// TIA Portal project "R1A-Cabi" (V15)

(* hardware
DEVICE "LINHA-DENIN"  ET 200S station
   slot 0: "Rack 0"  Rail
   slot 2: "IM151-8 PN/DP CPU"  IM151-8 CPU  6ES7 151-8AB00-0AB0  V2.7
      slot 1: "PROFINET-SLAVE"  PN-IO
         slot 1: "Port_1"  Port
         slot 2: "Port_2"  Port
         slot 3: "Port_3"  Port
   slot 4: "PM-E 24VDC_1"  PM-E 24VDC  6ES7 138-4CA01-0AA0
   slot 5: "DP interface_1"  DP  6ES7 138-4HA00-0AB0  V1.0
   slot 5: "8DI x 24VDC_1"  8DI x 24VDC  6ES7 131-4BF00-0AA0
   slot 6: "8DI x 24VDC_2"  8DI x 24VDC  6ES7 131-4BF00-0AA0
   slot 7: "8DI x 24VDC_3"  8DI x 24VDC  6ES7 131-4BF00-0AA0
   slot 8: "8DI x 24VDC_4"  8DI x 24VDC  6ES7 131-4BF00-0AA0
   slot 9: "8DO x 24VDC / 0.5A_1"  8DO x 24VDC / 0.5A  6ES7 132-4BF00-0AA0
   slot 10: "8DO x 24VDC / 0.5A_2"  8DO x 24VDC / 0.5A  6ES7 132-4BF00-0AA0
   slot 11: "8DO x 24VDC / 0.5A_3"  8DO x 24VDC / 0.5A  6ES7 132-4BF00-0AA0
   slot 12: "8DO x 24VDC / 0.5A_4"  8DO x 24VDC / 0.5A  6ES7 132-4BF00-0AA0
   slot 13: "8DO x 24VDC / 0.5A_5"  8DO x 24VDC / 0.5A  6ES7 132-4BF00-0AA0
   slot 14: "2AO x U ST_1"  2AO x U ST  6ES7 135-4FB01-0AB0
DEVICE "ET 200S station_1"  ET 200S station
   slot 0: "Rack_0"  Rail
   slot 0: "R2-REMOTA ENTRADA"  IM 151-3 PN  6ES7 151-3AA23-0AB0  V7.0
   slot 1: "PM-E 24VDC_1"  PM-E 24VDC  6ES7 138-4CA01-0AA0
   slot 2: "8DI x 24VDC_1"  8DI x 24VDC  6ES7 131-4BF00-0AA0
   slot 3: "8DI x 24VDC_2"  8DI x 24VDC  6ES7 131-4BF00-0AA0
   slot 4: "8DI x 24VDC_3"  8DI x 24VDC  6ES7 131-4BF00-0AA0
   slot 5: "8DI x 24VDC_4"  8DI x 24VDC  6ES7 131-4BF00-0AA0
   slot 6: "2AI x U ST_1"  2AI x U ST  6ES7 134-4FB01-0AB0
   slot 7: "2AI x U ST_2"  2AI x U ST  6ES7 134-4FB01-0AB0
   slot 8: "8DO x 24VDC / 0.5A_1"  8DO x 24VDC / 0.5A  6ES7 132-4BF00-0AA0
   slot 9: "8DO x 24VDC / 0.5A_2"  8DO x 24VDC / 0.5A  6ES7 132-4BF00-0AA0
   slot 10: "2AI x U ST_3"  2AI x U ST  6ES7 134-4FB01-0AB0
   slot 11: "2/4AI x RTD ST_1"  2/4AI x RTD ST  6ES7 134-4JB51-0AB0
   slot 12: "2/4AI x RTD ST_2"  2/4AI x RTD ST  6ES7 134-4JB51-0AB0
DEVICE "ET 200S station_2"  ET 200S station
   slot 0: "Rack_0"  Rail
   slot 0: "R3-REMOTA MESA DE COMANDO"  IM 151-3 PN  6ES7 151-3AA23-0AB0  V6.1
   slot 1: "PM-E 24VDC_1"  PM-E 24VDC  6ES7 138-4CA01-0AA0
   slot 2: "8DI x 24VDC_1"  8DI x 24VDC  6ES7 131-4BF00-0AA0
   slot 3: "8DI x 24VDC_2"  8DI x 24VDC  6ES7 131-4BF00-0AA0
   slot 4: "8DI x 24VDC_3"  8DI x 24VDC  6ES7 131-4BF00-0AA0
   slot 5: "2/4AI x RTD ST_1"  2/4AI x RTD ST  6ES7 134-4JB51-0AB0
   slot 6: "2/4AI x RTD ST_2"  2/4AI x RTD ST  6ES7 134-4JB51-0AB0
   slot 7: "2/4AI x RTD ST_3"  2/4AI x RTD ST  6ES7 134-4JB51-0AB0
   slot 8: "2/4AI x RTD ST_4"  2/4AI x RTD ST  6ES7 134-4JB51-0AB0
   slot 9: "2/4AI x RTD ST_5"  2/4AI x RTD ST  6ES7 134-4JB51-0AB0
   slot 10: "PM-E 24VDC_2"  PM-E 24VDC  6ES7 138-4CA01-0AA0
   slot 11: "2AI x U ST_1"  2AI x U ST  6ES7 134-4FB01-0AB0
   slot 12: "2AI x I 4WIRE ST_1"  2AI x I 4WIRE ST  6ES7 134-4GB11-0AB0
   slot 13: "2AI x I 4WIRE ST_2"  2AI x I 4WIRE ST  6ES7 134-4GB11-0AB0
   slot 14: "2AI x I 4WIRE ST_3"  2AI x I 4WIRE ST  6ES7 134-4GB11-0AB0
   slot 15: "8DO x 24VDC / 0.5A_1"  8DO x 24VDC / 0.5A  6ES7 132-4BF00-0AA0
   slot 16: "8DO x 24VDC / 0.5A_2"  8DO x 24VDC / 0.5A  6ES7 132-4BF00-0AA0
   slot 17: "8DO x 24VDC / 0.5A_3"  8DO x 24VDC / 0.5A  6ES7 132-4BF00-0AA0
   slot 18: "2AO x I ST_1"  2AO x I ST  6ES7 135-4GB01-0AB0
DEVICE "ET 200S station_3"  ET 200S station
   slot 0: "Rack_0"  Rail
   slot 0: "R4-REMOTA SAIDA"  IM 151-3 PN  6ES7 151-3AA23-0AB0  V6.1
   slot 1: "PM-E 24VDC_1"  PM-E 24VDC  6ES7 138-4CA01-0AA0
   slot 2: "8DI x 24VDC_1"  8DI x 24VDC  6ES7 131-4BF00-0AA0
   slot 3: "8DI x 24VDC_2"  8DI x 24VDC  6ES7 131-4BF00-0AA0
   slot 4: "8DI x 24VDC_3"  8DI x 24VDC  6ES7 131-4BF00-0AA0
   slot 5: "8DI x 24VDC_4"  8DI x 24VDC  6ES7 131-4BF00-0AA0
   slot 6: "2AI x U ST_1"  2AI x U ST  6ES7 134-4FB01-0AB0
   slot 7: "2AI x U ST_2"  2AI x U ST  6ES7 134-4FB01-0AB0
   slot 8: "2AI x U ST_3"  2AI x U ST  6ES7 134-4FB01-0AB0
   slot 9: "2AI x U ST_4"  2AI x U ST  6ES7 134-4FB01-0AB0
   slot 10: "2AI x U ST_5"  2AI x U ST  6ES7 134-4FB01-0AB0
   slot 11: "PM-E 24VDC_2"  PM-E 24VDC  6ES7 138-4CA01-0AA0
   slot 12: "2/4AI x RTD ST_1"  2/4AI x RTD ST  6ES7 134-4JB51-0AB0
   slot 13: "2/4AI x RTD ST_2"  2/4AI x RTD ST  6ES7 134-4JB51-0AB0
   slot 14: "2/4AI x RTD ST_3"  2/4AI x RTD ST  6ES7 134-4JB51-0AB0
   slot 15: "8DO x 24VDC / 0.5A_1"  8DO x 24VDC / 0.5A  6ES7 132-4BF00-0AA0
   slot 16: "2AO x I ST_1"  2AO x I ST  6ES7 135-4GB01-0AB0
   slot 17: "2AO x I ST_2"  2AO x I ST  6ES7 135-4GB01-0AB0
   slot 18: "2AO x I ST_3"  2AO x I ST  6ES7 135-4GB01-0AB0
   slot 19: "2AO x I ST_4"  2AO x I ST  6ES7 135-4GB01-0AB0
   slot 20: "2/4AI x RTD ST_4"  2/4AI x RTD ST  6ES7 134-4JB51-0AB0
   slot 21: "2/4AI x RTD ST_5"  2/4AI x RTD ST  6ES7 134-4JB51-0AB0
DEVICE "GSD device_1"  GSD.Device
   slot 0: "Rack_0"  Rail
DEVICE "GSD device_2"  GSD.Device
   slot 0: "Rack_0"  Rail
DEVICE "GSD device_3"  GSD.Device
   slot 0: "Rack_0"  Rail
DEVICE "GSD device_4"  GSD.Device
   slot 0: "Rack_0"  Rail
DEVICE "GSD device_5"  GSD.Device
   slot 0: "Rack_0"  Rail
DEVICE "GSD device_6"  GSD.Device
   slot 0: "Rack_0"  Rail
DEVICE "GSD device_7"  GSD.Device
   slot 0: "Rack_0"  Rail
DEVICE "GSD device_8"  GSD.Device
   slot 0: "Rack_0"  Rail
DEVICE "GSD device_9"  GSD.Device
   slot 0: "Rack_0"  Rail
DEVICE "GSD device_10"  GSD.Device
   slot 0: "Rack_0"  Rail
DEVICE "GSD device_11"  GSD.Device
   slot 0: "Rack_0"  Rail
DEVICE "GSD device_12"  GSD.Device
   slot 0: "Rack_0"  Rail
DEVICE "GSD device_13"  GSD.Device
   slot 0: "Rack_0"  Rail
DEVICE "GSD device_14"  GSD.Device
   slot 0: "Rack_0"  Rail
DEVICE "GSD device_15"  GSD.Device
   slot 0: "Rack_0"  Rail
*)

// ===== PLC "IM151-8 PN/DP CPU"  IM151-8 CPU =====

VAR_GLOBAL   // PLC tag table "Default tag table"
   "Tag_52" AT %T4 : Timer;
   "Tag_53" AT %M50.4 : Bool;
   "Tag_54" AT %T7 : Timer;
   "Tag_55" AT %M50.3 : Bool;
   "Tag_56" AT %MD0 : Real;
   "Tag_57" AT %M50.6 : Bool;
   "Tag_58" AT %MD5 : Real;
   "Tag_59" AT %M1.3 : Bool;
   "Tag_60" AT %M1.0 : Bool;
   "Tag_61" AT %M1.7 : Bool;
   "Tag_62" AT %MW22 : Word;
   "Tag_63" AT %M0.0 : Bool;
   "Tag_64" AT %MW32 : Word;
   "Tag_65" AT %MW34 : Word;
   "Tag_66" AT %MW36 : Word;
   "Tag_67" AT %T131 : Timer;
   "Tag_68" AT %T130 : Timer;
   "Tag_69" AT %M100.1 : Bool;
   "Tag_70" AT %T161 : Timer;
   "Tag_71" AT %T160 : Timer;
   "Tag_72" AT %T45 : Timer;
   "Tag_73" AT %T46 : Timer;
   "Tag_74" AT %T44 : Timer;
   "Tag_75" AT %M33.2 : Bool;
   "Tag_76" AT %M33.3 : Bool;
   "Tag_77" AT %M30.1 : Bool;
   "Tag_78" AT %M30.3 : Bool;
   "Tag_79" AT %M30.0 : Bool;
   "Tag_80" AT %M31.1 : Bool;
   "Tag_81" AT %M31.2 : Bool;
   "Tag_82" AT %M31.3 : Bool;
   "Tag_83" AT %M31.4 : Bool;
   "Tag_84" AT %MW30 : Word;
   "Tag_85" AT %T40 : Timer;
   "Tag_86" AT %T41 : Timer;
   "Tag_87" AT %T42 : Timer;
   "Tag_88" AT %M33.0 : Bool;
   "Tag_89" AT %M33.1 : Bool;
   "Tag_90" AT %M33.4 : Bool;
   "Tag_91" AT %M33.5 : Bool;
   "Tag_92" AT %M31.0 : Bool;
   "Tag_93" AT %M30.2 : Bool;
   "Tag_94" AT %T20 : Timer;
   "Tag_95" AT %T21 : Timer;
   "Tag_96" AT %T22 : Timer;
   "Tag_97" AT %T23 : Timer;
   "Tag_98" AT %T48 : Timer;
   "Tag_99" AT %M26.0 : Bool;
   "Tag_100" AT %M26.1 : Bool;
   "Tag_101" AT %M51.3 : Bool;
   "Tag_102" AT %M100.0 : Bool;
   "Tag_103" AT %M100.3 : Bool;
   "Tag_104" AT %M100.5 : Bool;
   "Tag_105" AT %M10.3 : Bool;
   "Tag_106" AT %M60.7 : Bool;
   "Tag_107" AT %MD18 : Real;
   "Tag_108" AT %M50.7 : Bool;
END_VAR

VAR_GLOBAL   // PLC tag table "STEP7 classic symbols"
   "Q206" AT %Q20.6 : Bool;   // R2 - PROGRAMADOR CHAMA 2
   "Q205" AT %Q20.5 : Bool;   // R2 - PROGRAMADOR CHAMA 1
   "Q204" AT %Q20.4 : Bool;   // R2 - SEGURANCA CHAMUS
   "Q203" AT %Q20.3 : Bool;   // R2 - LIBERA GAS QUEIMADORES 1 E 3
   "I407" AT %I40.7 : Bool;   // R4 - LIGA MAQUINA
   "I406" AT %I40.6 : Bool;   // R4 - TROCA ROLO ER
   "I405" AT %I40.5 : Bool;   // R4 - INDEP/SINC ER
   "I404" AT %I40.4 : Bool;   // R4 - JOG ER
   "I403" AT %I40.3 : Bool;   // R4 - DESLIGA ER
   "I402" AT %I40.2 : Bool;   // R4 - LIGA / SINCR ER
   "I401" AT %I40.1 : Bool;   // R4 - BALANCA SUPERIOR ER
   "I400" AT %I40.0 : Bool;   // R4 - BALANCA INFERIOR ER
   "I412" AT %I41.2 : Bool;   // R4 - BALANCA SECADEIRA 2
   "I411" AT %I41.1 : Bool;   // R4 - BALANCA ESTICADOR
   "I410" AT %I41.0 : Bool;   // R4 - BALANCA SECADEIRA 1
   "I417" AT %I41.7 : Bool;   // R4 - GERA PULSO SAIDA ESTICADOR
   "I416" AT %I41.6 : Bool;   // R4 - GERA PULSO ENT ESTICADOR
   "I415" AT %I41.5 : Bool;   // R4 - BALANCA PUXADOR JOTA SAIDA
   "I414" AT %I41.4 : Bool;   // R4 - BALANCA SECADEIRA 4
   "I413" AT %I41.3 : Bool;   // R4 - BALANCA SECADEIRA 3
   "I427" AT %I42.7 : Bool;   // R4 - - VELOCIDADE
   "I426" AT %I42.6 : Bool;   // R4 - EMERGENCIA
   "I425" AT %I42.5 : Bool;   // R4 - + VELOCIDADE
   "I424" AT %I42.4 : Bool;   // R4 - DESLIGA MAQUINA
   "P_QW102" AT %QW102 : Int;   // R1A - REFERENCIA INVERSOR RESERVA 2
   "P_QW100" AT %QW100 : Int;   // R1A - REFERENCIA INVERSOR RESERVA 1
   "I304" AT %I30.4 : Bool;   // R3 - - VELOCIDADE
   "I303" AT %I30.3 : Bool;   // R3 - + VELOCIDADE
   "I302" AT %I30.2 : Bool;   // R3 - EMERGENCIA
   "I301" AT %I30.1 : Bool;   // R3 - DESLIGA MAQUINA
   "I300" AT %I30.0 : Bool;   // R3 - LIGA MAQUINA
   "I307" AT %I30.7 : Bool;   // R3 - DESTRAVA ALARME
   "I306" AT %I30.6 : Bool;   // R3 - TRAVA BALACIM
   "I305" AT %I30.5 : Bool;   // R3 - JOG GERAL
   "I317" AT %I31.7 : Bool;   // R3 - NIVEL TQ 2 NEUTRALIZACAO 2
   "I316" AT %I31.6 : Bool;   // R3 - NIVEL TQ 1 NEUTRALIZACAO 2
   "I315" AT %I31.5 : Bool;   // R3 - NIVEL TQ 2 LAVAGEM 1
   "I314" AT %I31.4 : Bool;   // R3 - NIVEL TQ 1 LAVAGEM 1
   "I313" AT %I31.3 : Bool;   // R3 - NIVEL TQ 2 NEUTRALIZACAO 1
   "I312" AT %I31.2 : Bool;   // R3 - NIVEL TQ 1 NEUTRALIZACAO 1
   "I311" AT %I31.1 : Bool;   // R3 - IGNICAO
   "I310" AT %I31.0 : Bool;   // R3 - IGNICAO MANUAL
   "I324" AT %I32.4 : Bool;   // R3 - ACIONA ALARME
   "I323" AT %I32.3 : Bool;   // R3 - PRESSOSTADO GERAL AR
   "I322" AT %I32.2 : Bool;   // R3 - TERMICO BOMBA 3
   "I321" AT %I32.1 : Bool;   // R3 - NIVEL TQ 2 LAVAGEM 2
   "I320" AT %I32.0 : Bool;   // R3 - NIVEL TQ 1 LAVAGEM 2
   "I327" AT %I32.7 : Bool;   // R3 - RESERVA
   "I107" AT %I10.7 : Bool;   // R1A - TERM COLETOR PO 1 CHAMUS
   "I106" AT %I10.6 : Bool;   // R1A - TERM EXAUSTOR CHAMUS
   "I105" AT %I10.5 : Bool;   // R1A - TERM ESCOVA 4 CHAMUS
   "I104" AT %I10.4 : Bool;   // R1A - TERM ESCOVA 3 CHAMUS
   "I103" AT %I10.3 : Bool;   // R1A - TERM ESCOVA 2 CHAMUS
   "I102" AT %I10.2 : Bool;   // R1A - TERM ESCOVA 1 CHAMUS
   "I101" AT %I10.1 : Bool;   // R1A - TERM VENTILADOR RAPIDO CHAMUS
   "I100" AT %I10.0 : Bool;   // R1A - TERM VENTILADOR LENTO CHAMUS
   "I116" AT %I11.6 : Bool;   // R1A - TERM EXAUSTOR SECADEIRA 1
   "I115" AT %I11.5 : Bool;   // R1A - TERM UNIDADE SKIW DIREITO
   "I114" AT %I11.4 : Bool;   // R1A - TERM UNIDADE SKIW ESQUERDO
   "I113" AT %I11.3 : Bool;   // R1A - TERM ENTORTADOR TRAMA PARALELO
   "I112" AT %I11.2 : Bool;   // R1A - TERM ENTORTADOR CURVO
   "I111" AT %I11.1 : Bool;   // R1A - TERM ROSCA FOULARD
   "I110" AT %I11.0 : Bool;   // R1A - TERM COLETOR PO 2 CHAMUS
   "I117" AT %I11.7 : Bool;   // R1A - TERM EXAUSTOR SECADEIRA 2
   "I127" AT %I12.7 : Bool;   // R1A - TERM CILINDROS EXTRACTA LAV 2
   "I126" AT %I12.6 : Bool;   // R1A - TERM CILINDROS EXTRACTA LAV 1
   "I125" AT %I12.5 : Bool;   // R1A - RESERVA
   "I124" AT %I12.4 : Bool;   // R1A - RESERVA
   "I123" AT %I12.3 : Bool;   // R1A - TERM EXAUSTOR NEUTRALIZACAO 2
   "I122" AT %I12.2 : Bool;   // R1A - TERM EXAUSTOR NEUTRALIZACAO 1
   "I121" AT %I12.1 : Bool;   // R1A - TERM EXAUSTOR SECADEIRA 4
   "I120" AT %I12.0 : Bool;   // R1A - TERM EXAUSTOR SECADEIRA 3
   "Q303" AT %Q30.3 : Bool;   // R3 - ALARME
   "Q302" AT %Q30.2 : Bool;   // R3 - DESTRAVA ALARME
   "Q301" AT %Q30.1 : Bool;   // R3 - TRAVA BALANCIM
   "Q300" AT %Q30.0 : Bool;   // R3 - MAQUINA LIGADA
   "Q312" AT %Q31.2 : Bool;   // R3 - AGUA LIMPA FITRO ROTATIVO NEUTRALIZACAO 1
   "Q311" AT %Q31.1 : Bool;   // R3 - VAZAO AGUA NEUTRALIZACAO 2
   "Q310" AT %Q31.0 : Bool;   // R3 - VAZAO AGUA NEUTRALIZACAO 1
   "Q317" AT %Q31.7 : Bool;   // R3 - RESERVA
   "Q316" AT %Q31.6 : Bool;   // R3 - RESERVA
   "Q315" AT %Q31.5 : Bool;   // R3 - AGUA TROCADOR CALOR NEUTRALIZACAO 2
   "Q314" AT %Q31.4 : Bool;   // R3 - AGUA TROCADOR CALOR NEUTRALIZACAO 1
   "Q313" AT %Q31.3 : Bool;   // R3 - AGUA LIMPA FITRO ROTATIVO NEUTRALIZACAO 2
   "Q327" AT %Q32.7 : Bool;   // R3 - RESERVA
   "Q326" AT %Q32.6 : Bool;   // R3 - RESERVA
   "Q325" AT %Q32.5 : Bool;   // R3 - RESERVA
   "Q324" AT %Q32.4 : Bool;   // R3 - BOMBA 3
   "Q323" AT %Q32.3 : Bool;   // R3 - TEMPERATURA 2 LAVAGEM 2
   "Q322" AT %Q32.2 : Bool;   // R3 - TEMPERATURA 1 LAVAGEM 2
   "Q321" AT %Q32.1 : Bool;   // R3 - TEMPERATURA 2 LAVAGEM 1
   "Q320" AT %Q32.0 : Bool;   // R3 - TEMPERATURA 1 LAVAGEM 1
   "P_PQW302" AT %QW302 : Word;   // R3 - VALVULA TROCADOR CALOR 2
   "P_PQW300" AT %QW300 : Word;   // R3 - VALVULA TROCADOR CALOR 1
   "I200" AT %I20.0 : Bool;   // R2 - PRESSOSTATO VENTILADOR CHAMUS
   "I207" AT %I20.7 : Bool;   // R2 - FOTOCELULA DETETORA TECIDO CHAMUS
   "I423" AT %I42.3 : Bool;   // R4 - GERA PULSO SAIDA SKIW DIREITO
   "I422" AT %I42.2 : Bool;   // R4 - GERA PULSO SAIDA SKIW ESQUERDO
   "I421" AT %I42.1 : Bool;   // R4 - GERA PULSO ENT SKIW DIREITO
   "I420" AT %I42.0 : Bool;   // R4 - NIVEL DO FOULARD
   "I432" AT %I43.2 : Bool;   // R4 - ENTORTADOR TRAMA PARALELO AVANCADO
   "I431" AT %I43.1 : Bool;   // R4 - TRAVA BALANCIM
   "I430" AT %I43.0 : Bool;   // R4 - ACIONA ALARME
   "I437" AT %I43.7 : Bool;   // R4 - SKIW ESQUERDO RECUADO
   "I436" AT %I43.6 : Bool;   // R4 - SKIW ESQUERDO AVANCADO
   "I435" AT %I43.5 : Bool;   // R4 - SKIW DIREITO RECUADO
   "I434" AT %I43.4 : Bool;   // R4 - SKIW DIREITO AVANCADO
   "I433" AT %I43.3 : Bool;   // R4 - ENTORTADOR TRAMA PARALELO RECUADO
   "P_PIW402" AT %IW402 : Int;   // R4 - VELOCIDADE IND TROCA ROLO ER
   "P_PIW400" AT %IW400 : Int;   // R4 - BALANCA ER
   "P_PIW406" AT %IW406 : Int;   // R4 - BALANCA ESTICADOR
   "P_PIW404" AT %IW404 : Int;   // R4 - BALANCA SECADEIRA 1
   "P_PIW410" AT %IW410 : Int;   // R4 - BALANCA SECADEIRA 3
   "P_PIW408" AT %IW408 : Int;   // R4 - BALANCA SECADEIRA 2
   "P_PIW414" AT %IW414 : Int;   // R4 - BALANCA PUX JOTA SAIDA
   "P_PIW412" AT %IW412 : Int;   // R4 - BALANCA SECADEIRA 4
   "P_PIW418" AT %IW418 : Word;   // R4 - RESERVA
   "P_PIW416" AT %IW416 : Int;   // R4 - MEDIDOR UMIDADE
   "P_PIW428" AT %IW428 : Int;   // R4 - TEMPERATURA SECADEIRA 4
   "P_PIW430" AT %IW430 : Word;   // R4 - RESERVA
   "Q127" AT %Q12.7 : Bool;   // R1A - EXAUSTOR NEUTRALIZACAO 2
   "Q126" AT %Q12.6 : Bool;   // R1A - horime
   "Q125" AT %Q12.5 : Bool;   // R1A - EXAUSTOR NEUTRALIZACAO 1
   "Q124" AT %Q12.4 : Bool;   // R1A - EXAUSTOR SECADEIRA 4
   "Q123" AT %Q12.3 : Bool;   // R1A - EXAUSTOR SECADEIRA 3
   "Q122" AT %Q12.2 : Bool;   // R1A - RECUA UNIDADE SKIW DIREITO
   "Q121" AT %Q12.1 : Bool;   // R1A - EXAUSTOR SECADEIRA 2
   "Q120" AT %Q12.0 : Bool;   // R1A - AVANCA UNIDADE SKIW DIREITO
   "Q136" AT %Q13.6 : Bool;   // R1A - RESERVA
   "Q135" AT %Q13.5 : Bool;   // R1A - DESBLOQUEIO FRENTE RESERVA 2
   "Q134" AT %Q13.4 : Bool;   // EXAUSTOR 2 DA IMPREGNAÇÃO - NEUTRALIZAÇÃO
   "Q133" AT %Q13.3 : Bool;   // R1A - RESERVA
   "Q132" AT %Q13.2 : Bool;   // R1A - RESERVA
   "Q131" AT %Q13.1 : Bool;   // R1A - EMERGENCIA
   "Q130" AT %Q13.0 : Bool;   // R1A - VALVULA DE ÁGUA
   "Q137" AT %Q13.7 : Bool;   // R1A - RESERVA
   "Q147" AT %Q14.7 : Bool;   // R1A - RESERVA
   "Q146" AT %Q14.6 : Bool;   // R1A - RESERVA
   "Q145" AT %Q14.5 : Bool;   // R1A - RESERVA
   "Q144" AT %Q14.4 : Bool;   // R1A - RESERVA
   "Q143" AT %Q14.3 : Bool;   // R1A - FILTRO ROTATIVO NEUTRALIZACAO 1
   "Q142" AT %Q14.2 : Bool;   // R1A - BOMBA CIRC NEUTRALIZACAO 2
   "Q141" AT %Q14.1 : Bool;   // R1A - FILTRO ROTATIVO NEUTRALIZACAO 1
   "Q140" AT %Q14.0 : Bool;   // R1A - BOMBA CIRC NEUTRALIZACAO 1
   "P_PIW438" AT %IW438 : Int;   // R4 - TEMPERATURA TANQUE 4 PRODUTO
   "P_PIW436" AT %IW436 : Int;   // R4 - TEMPERATURA TANQUE 3 PRODUTO
   "P_PIW434" AT %IW434 : Int;   // R4 - TEMPERATURA TANQUE 2 PRODUTO
   "P_PIW432" AT %IW432 : Int;   // R4 - TEMPERATURA TANQUE 1 PRODUTO
   "T30" AT %T30 : Timer;   // R4 - TEMPO PARA ABRE/FECHA VALVULA DE NIVEL CX DE GOMA
   "T31" AT %T31 : Timer;   // R4 - TEMPO PARA ALARME DE NIVEL CX DE GOMA
   "T50" AT %T50 : Timer;   // TEMP RETARDO DESLIGA MQ R3
   "M40.0" AT %M40.0 : Bool;   // RETARDO DESLIGA MQ R3
   "M38.3" AT %M38.3 : Bool;   // SANFOR - ALARME DESLIGA MAQUIMA
   "M38.2" AT %M38.2 : Bool;   // R4 - ALARME DESLIGA MAQUIMA
   "M38.1" AT %M38.1 : Bool;   // R3 - ALARME DESLIGA MAQUIMA
   "M38.0" AT %M38.0 : Bool;   // R2 - ALARME DESLIGA MAQUIMA
   "MW38" AT %MW38 : Word;   // WORD DE ALARME DESLIGA MAQUINA
   "M51.0" AT %M51.0 : Bool;   // ALARMES DE TEMPERATURA
   "P_PIW422" AT %IW422 : Word;   // R4 - Temperatura do Foulard FV210
   "P_PIW420" AT %IW420 : Int;   // R4 - TEMPERATURA SECADEIRA 1
   "P_PIW426" AT %IW426 : Int;   // R4 - TEMPERATURA SECADEIRA 3
   "P_PIW424" AT %IW424 : Int;   // R4 - TEMPERATURA SECADEIRA 2
   "Q407" AT %Q40.7 : Bool;   // R4 - ALARME DE NIVEL BAIXO CAIXA DE GOMA
   "Q406" AT %Q40.6 : Bool;   // R4 - VALVULA PRODUTO FOULARD
   "Q405" AT %Q40.5 : Bool;   // R4 - TQ4_PRD
   "Q404" AT %Q40.4 : Bool;   // R4 - TQ3_PRD
   "Q403" AT %Q40.3 : Bool;   // R4 - TQ2_PRD
   "Q402" AT %Q40.2 : Bool;   // R4 - TQ1_PRD
   "Q401" AT %Q40.1 : Bool;   // R4 - ER LIGADO
   "Q400" AT %Q40.0 : Bool;   // R4 - TROCA ROLO ER
   "P_PQW402" AT %QW402 : Word;   // R4 - VALVULA FLUXO AGUA CX1
   "P_PQW400" AT %QW400 : Word;   // R4 - VALVULA SECADEIRA 1
   "P_PQW404" AT %QW404 : Word;   // R4 - VALVULA SECADEIRA 2
   "P_PQW406" AT %QW406 : Word;   // R4 - VALVULA SECADEIRA 3
   "P_PQW410" AT %QW410 : Word;   // R4 - VALVULA FLUXO AGUA CX2
   "P_PQW408" AT %QW408 : Word;   // R4 - VALVULA SECADEIRA 4
   "P_PQW414" AT %QW414 : Word;   // R4 - RESERVA
   "P_PQW412" AT %QW412 : Word;   // R4 - RESERVA
   "I326" AT %I32.6 : Bool;   // R3 - RESERVA
   "I325" AT %I32.5 : Bool;   // R3 - RESERVA
   "P_PIW302" AT %IW302 : Int;   // R3 - RESERVA
   "P_PIW300" AT %IW300 : Int;   // R3 - TEMP NEUTRALIZACAO 1
   "P_PIW306" AT %IW306 : Int;   // R3 - TEMP TQ 2 LAVAGEM 1
   "P_PIW304" AT %IW304 : Int;   // R3 - TEMP TQ 1 LAVAGEM 1
   "P_PIW310" AT %IW310 : Int;   // R3 - RESERVA
   "P_PIW308" AT %IW308 : Int;   // R3 - TEMP NEUTRALIZACAO 2
   "P_PIW314" AT %IW314 : Int;   // R3 - TEMP TQ 2 LAVAGEM 2
   "P_PIW312" AT %IW312 : Int;   // R3 - TEMP TQ 1 LAVAGEM 2
   "P_PIW318" AT %IW318 : Int;   // R3 - BALANCIM NEUTRALIZACAO 1
   "P_PIW316" AT %IW316 : Int;   // R3 - BALANCIM LAVAGEM 1
   "P_PIW322" AT %IW322 : Int;   // R3 - BALANCIM LAVAGEM 2
   "P_PIW320" AT %IW320 : Int;   // R3 - BALANCIM NEUTRALIZACAO 2
   "P_PIW324" AT %IW324 : Word;   // R3 - MEDIDOR VAZAO NEUTRALIZACAO 1
   "P_PIW326" AT %IW326 : Word;   // R3 - MEDIDOR VAZAO NEUTRALIZACAO 2
   "P_PIW330" AT %IW330 : Int;   // R3 - CELULA CARGA EXTRACTA 2
   "P_PIW328" AT %IW328 : Int;   // R3 - CELULA CARGA EXTRACTA 1
   "P_PIW334" AT %IW334 : Word;   // R3 - RESERVA
   "P_PIW332" AT %IW332 : Int;   // R3 - SENSOR PH
   "Q307" AT %Q30.7 : Bool;   // R3 - NIVEL TQ 2 NEUTRALIZACAO 2
   "Q306" AT %Q30.6 : Bool;   // R3 - NIVEL TQ 1 NEUTRALIZACAO 2
   "Q305" AT %Q30.5 : Bool;   // R3 - NIVEL TQ 2 NEUTRALIZACAO 1
   "Q304" AT %Q30.4 : Bool;   // R3 - NIVEL TQ 1 NEUTRALIZACAO 1
   "I235" AT %I23.5 : Bool;   // R2 - RESERVA
   "I234" AT %I23.4 : Bool;   // R2 - - VELOCIDADE
   "I233" AT %I23.3 : Bool;   // R2 - + VELOCIDADE
   "I232" AT %I23.2 : Bool;   // R2 - EMERGENCIA
   "I231" AT %I23.1 : Bool;   // R2 - DESLIGA MAQUINA
   "I230" AT %I23.0 : Bool;   // R2 - LIGA MAQUINA
   "P_PIW200" AT %IW200 : Int;   // R2 - BALANCA PUX JOTA ENT
   "P_PIW202" AT %IW202 : Int;   // R2 - VELOCIDADE IND TROCA ROLO PUX
   "P_PIW206" AT %IW206 : Word;   // R2 - RESERVA
   "P_PIW204" AT %IW204 : Int;   // R2 - SENSOR BALANCIM CHAMUS
   "Q217" AT %Q21.7 : Bool;   // R2 - RESERVA
   "Q216" AT %Q21.6 : Bool;   // R2 - PUXADOR JOTA ENT LIGADO
   "Q215" AT %Q21.5 : Bool;   // R2 - RESERVA
   "Q214" AT %Q21.4 : Bool;   // R2 - TROCA ROLO PUX JOTA ENT
   "Q213" AT %Q21.3 : Bool;   // R2 - RESERVA
   "Q212" AT %Q21.2 : Bool;   // R2 - SERVO 1 FECHA
   "Q211" AT %Q21.1 : Bool;   // R2 - SERVO 1 ABRE
   "Q210" AT %Q21.0 : Bool;   // R2 - PROGRAMADOR CHAMA 4
   "P_PQW202" AT %QW202 : Word;   // R2 - RESERVA
   "P_PQW200" AT %QW200 : Word;   // R2 - RESERVA
   "Q202" AT %Q20.2 : Bool;   // R2 - LIBERA GAS QUEIMADORES 2 E 4
   "Q201" AT %Q20.1 : Bool;   // R2 - POSICAO CHAMA AR-2
   "Q200" AT %Q20.0 : Bool;   // R2 - POSICAO CHAMA AR-1
   "Q207" AT %Q20.7 : Bool;   // R2 - PROGRAMADOR CHAMA 3
   "I136" AT %I13.6 : Bool;   // R1A - RESERVA
   "I135" AT %I13.5 : Bool;   // R1A - TERM BOMBA CIRC NEUTRALIZACAO 2
   "I134" AT %I13.4 : Bool;   // R1A - RESERVA
   "I133" AT %I13.3 : Bool;   // R1A - TERM FILTRO ROTATIVO NEUTRALIZACAO 1
   "I132" AT %I13.2 : Bool;   // R1A - PROTECAO INVERSOR RESERVA 2
   "I131" AT %I13.1 : Bool;   // R1A - TERM BOMBA CIRC NEUTRALIZACAO 1
   "I130" AT %I13.0 : Bool;   // R1A - PROTECAO INVERSOR RESERVA 1
   "I137" AT %I13.7 : Bool;   // R1A - TERM FILTRO ROTATIVO NEUTRALIZACAO 2
   "Q107" AT %Q10.7 : Bool;   // R1A - COLETOR PO 2 CHAMUS
   "Q106" AT %Q10.6 : Bool;   // R1A - COLETOR PO 1 CHAMUS
   "Q105" AT %Q10.5 : Bool;   // R1A - EXAUSTOR CHAMUS
   "Q104" AT %Q10.4 : Bool;   // R1A - RAPIDO VENTILADOR CHAMUS
   "Q103" AT %Q10.3 : Bool;   // R1A - ESCOVAS 3 E 4 CHAMUS
   "Q102" AT %Q10.2 : Bool;   // R1A - LENTO VENTILADOR CHAMUS
   "Q101" AT %Q10.1 : Bool;   // R1A - ESCOVAS 1 E 2 CHAMUS
   "Q100" AT %Q10.0 : Bool;   // R1A - AUXILIAR RAPIDO VENTILADOR CHAMUS
   "Q116" AT %Q11.6 : Bool;   // R1A - RECUA UNIDADE SKIW ESQUERDO
   "Q115" AT %Q11.5 : Bool;   // R1A - AVANCA ENTORTADOR TRAMA PARALELO
   "Q114" AT %Q11.4 : Bool;   // R1A - AVANCA UNIDADE SKIW ESQUERDO
   "Q113" AT %Q11.3 : Bool;   // R1A - RECUA ENTORTADOR TRAMA CURVO
   "Q112" AT %Q11.2 : Bool;   // R1A - EXAUSTOR SECADEIRA 1
   "Q111" AT %Q11.1 : Bool;   // R1A - AVANCA ENTORTADOR TRAMA CURVO
   "Q110" AT %Q11.0 : Bool;   // R1A - ROSCA FOULARD
   "Q117" AT %Q11.7 : Bool;   // R1A - RECUA ENTORTADOR TRAMA PARALELO
   "T3" AT %T3 : Timer;   // TEMPO DO AUDIO ANTES DA PARTIDA
   "M12_0" AT %M12.0 : Bool;   // AUXILIAR SINALIZAÇÃO AUDIO LIGA
   "T1" AT %T1 : Timer;   // TEMPO DE RESET DOS ALARMES NA ENERGIZAÇÃO DO PLC
   "T2" AT %T2 : Timer;   // TEMPO DE RESET DOS INVERSORES
   "M11_0" AT %M11.0 : Bool;   // AUXILIAR RESET DOS ALARMES
   "M10_0" AT %M10.0 : Bool;   // AUXILIAR - LIGA MÁQUINA
   "I206" AT %I20.6 : Bool;   // R2 - NIVEIS DE AGUA Q1/Q2/Q3/Q4
   "I205" AT %I20.5 : Bool;   // R2 - SERVO AR/GAS ABERTO
   "I204" AT %I20.4 : Bool;   // R2 - TERMOSTATOS Q1/Q2/Q3/Q4
   "I203" AT %I20.3 : Bool;   // R2 - SERVO AR/GAS FECHADO
   "I202" AT %I20.2 : Bool;   // R2 - PRESSOSTATO GAS PRESSAO ALTA/BAIXA
   "I201" AT %I20.1 : Bool;   // R2 - PRESSOSTATO CHAMUS
   "I217" AT %I21.7 : Bool;   // R2 - FALHA CHAMA QUEIMADOR 4
   "I216" AT %I21.6 : Bool;   // R2 - FALHA CHAMA QUEIMADOR 3
   "I215" AT %I21.5 : Bool;   // R2 - FALHA CHAMA QUEIMADOR 2
   "I214" AT %I21.4 : Bool;   // R2 - FALHA CHAMA QUEIMADOR 1
   "I213" AT %I21.3 : Bool;   // R2 - LIBERA GAS QUEIMADOR 4
   "I212" AT %I21.2 : Bool;   // R2 - LIBERA GAS QUEIMADOR 3
   "I211" AT %I21.1 : Bool;   // R2 - LIBERA GAS QUEIMADOR 2
   "I210" AT %I21.0 : Bool;   // R2 - LIBERA GAS QUEIMADOR 1
   "I220" AT %I22.0 : Bool;   // R2 - BALANCA INFERIOR JOTA ENT
   "I227" AT %I22.7 : Bool;   // R2 - ACIONA ALARME
   "I226" AT %I22.6 : Bool;   // R2 - TROCA ROLO PUXADOR JOTA ENT
   "I225" AT %I22.5 : Bool;   // R2 - INDEP/SINCR PUXADOR JOTA ENT
   "I224" AT %I22.4 : Bool;   // R2 - JOG PUXADOR JOTA ENT
   "I223" AT %I22.3 : Bool;   // R2 - DESLIGA PUXADOR JOTA ENT
   "I222" AT %I22.2 : Bool;   // R2 - LIGA/SINCR PUXADOR JOTA ENT
   "I221" AT %I22.1 : Bool;   // R2 - BALANCA SUPERIOR JOTA ENT
   "I237" AT %I23.7 : Bool;   // R2 - TRAVA BALANCIM
   "I236" AT %I23.6 : Bool;   // R2 - RESERVA
   "Tag_1" AT %MW0 : Word;
   "Tag_2" AT %EW1000 : Word;
   "Tag_3" AT %AW1000 : Word;
   "Tag_4" AT %AW1002 : Word;
   "Tag_5" AT %EW1020 : Word;
   "Tag_6" AT %AW1020 : Word;
   "Tag_7" AT %AW1022 : Word;
   "Tag_8" AT %EW1040 : Word;
   "Tag_9" AT %AW1040 : Word;
   "Tag_10" AT %AW1042 : Word;
   "Tag_11" AT %EW1060 : Word;
   "Tag_12" AT %AW1060 : Word;
   "Tag_13" AT %AW1062 : Word;
   "Tag_14" AT %EW1080 : Word;
   "Tag_15" AT %AW1080 : Word;
   "Tag_16" AT %AW1082 : Word;
   "Tag_17" AT %EW1120 : Word;
   "Tag_18" AT %AW1120 : Word;
   "Tag_19" AT %AW1122 : Word;
   "Tag_20" AT %EW1140 : Word;
   "Tag_21" AT %AW1140 : Word;
   "Tag_22" AT %AW1142 : Word;
   "Tag_23" AT %EW212 : Word;
   "Tag_24" AT %EW214 : Word;
   "Tag_25" AT %EW216 : Word;
   "Tag_26" AT %EW218 : Word;
   "Tag_27" AT %EW1160 : Word;
   "Tag_28" AT %AW1160 : Word;
   "Tag_29" AT %AW1162 : Word;
   "Tag_30" AT %EW1180 : Word;
   "Tag_31" AT %AW1180 : Word;
   "Tag_32" AT %AW1182 : Word;
   "Tag_33" AT %EW1200 : Word;
   "Tag_34" AT %AW1200 : Word;
   "Tag_35" AT %AW1202 : Word;
   "Tag_36" AT %EW1240 : Word;
   "Tag_37" AT %AW1240 : Word;
   "Tag_38" AT %AW1242 : Word;
   "Tag_39" AT %EW1260 : Word;
   "Tag_40" AT %AW1260 : Word;
   "Tag_41" AT %AW1262 : Word;
   "Tag_42" AT %EW1280 : Word;
   "Tag_43" AT %AW1280 : Word;
   "Tag_44" AT %AW1282 : Word;
   "Tag_45" AT %EW1300 : Word;
   "Tag_46" AT %AW1300 : Word;
   "Tag_47" AT %AW1302 : Word;
   "Tag_48" AT %EW1320 : Word;
   "Tag_49" AT %AW1320 : Word;
   "Tag_50" AT %AW1322 : Word;
   "Tag_51" AT %MW42 : Word;
END_VAR

DATA_BLOCK "DB PRINCIPAL"   // DB1
TITLE = Automation Pack Automação Indl. e Com. Ltda.
{ S7_Optimized_Access := 'FALSE' }
AUTHOR : THALLES
FAMILY : MAIN
NAME : LINHA1
VERSION : 0.1
// Cliente: Texima S/A Ind. de Máquinas
// Cliente Final: Cia. Fiação e Tecidos Santo Antonio.
// Máquina: Linha 1 DENIN - O.S.: 24.626
   VAR
      AUXILIARES : Struct   // AUXILIARES - PRINCIPAL DE USO GERAL
         SEMPRE_0 : Bool;   // BIT SEMPRE DESLIGADO - "0"
         SEMPRE_1 : Bool := TRUE;   // BIT SEMPRE LIGADO - "1"
         RESERVA_02 : Bool;   // RESERVA
         RESERVA_03 : Bool;   // RESERVA
         RESERVA_04 : Bool;   // RESERVA
         RESERVA_05 : Bool;   // RESERVA
         RESERVA_06 : Bool;   // RESERVA
         RESERVA_07 : Bool;   // RESERVA
         BASE_1_SCAN : Bool := TRUE;   // BIT QUE ALTERA SEU VALOR A CADA SCAN
         BASE_100MS : Bool;   // BIT QUE ALTERA SEU VALOR A CADA 50MS - PERIODO=100MS
         BASE_500MS : Bool := TRUE;   // BIT QUE ALTERA SEU VALOR A CADA 250MS - PERIODO=500MS
         BASE_1S : Bool := TRUE;   // BIT QUE ALTERA SEU VALOR A CADA 500MS - PERIODO=1S
      END_STRUCT;
      ALARME : Struct
         EMERGENCIA_GERAL : Bool;
         PRESSOSTATO_GERAL : Bool;
         INV_RESERVA1 : Bool;
         INV_RESERVA2 : Bool;
      END_STRUCT;
      COMANDOS : Struct   // COMANDOS
         ALARME_ALTO : Bool := TRUE;   // BIT QUE INDICA QUE ALGUM ALARME DE NIVEL ALTO FOI GERADO
         ALARME_BAIXO : Bool := TRUE;   // BIT QUE INDICA QUE ALGUM ALARME DE NIVEL BAIXO FOI GERADO
         JOG : Bool;   // 1=JOG GERAL
         MARCHA : Bool;   // 1=MÁQUINA LIGADA
         AUX_JOG : Bool;
         AUX_MARCHA : Bool;
         RESET_INVERSORES : Bool;   // RESET DOS ALARMES DOS INVERSORES - QUANDO EM 1 RESET DOS ALARMES DOS INVERSORES
         RESET_ALARMES : Bool;   // RESET DOS ALARMES DA MÁQUINA - QUANDO EM 1 RESET TODOS OS ALARMES
         BOTAO_EMERGENCIA : Bool := TRUE;   // BIT COMANDO DOS BOTÕES EMERGENCIA
         BOTAO_DESLIGA : Bool := TRUE;   // BIT COMANDO DOS BOTÕES DESLIGA
         BOTAO_JOG : Bool;   // BIT COMANDO DOS BOTÕES JOG
         BOTAO_LIGA : Bool;   // BIT COMANDO DOS BOTÕES LIGA
         BOTAO_INC_VEL : Bool;   // BIT COMANDO DOS BOTÕES + VEL
         BOTAO_DEC_VEL : Bool;   // BIT COMANDO DOS BOTÕES - VEL
         PARTIDA_MARCHA_SIN : Bool;
         PARTIDA_JOG_SIN : Bool;
         MOTOR_SELECIONADO : Bool := TRUE;   // 1=ALGUM MOTOR DE TRAÇÃO ESTÁ SELECIONADO
         BALANCA_FORA_POSICAO : Bool;   // 1=INDICAÇÃO DE BALANÇA FORA DE POSIÇÃO
         BALANCA_TRAVA : Bool;   // 1=TRAVA OS ALARMES DE BALANCIM DA MÁQUINA
         BOTAO_TRAVA_BALANCA : Bool;   // BIT COMANDO DOS BOTÕES TRAVA BALACIM
         COMANDO_REC_ALARME : Bool;   // BIT COMANDO RECONHECE ALARME
         SIRENE_LIGA : Bool;   // ACIONA SIRENE QUANDO LIGA A MAQUINA
         RESERVA2_6 : Bool;   // RESERVA
         RESERVA2_7 : Bool;   // RESERVA
         INV_RESERVA1 : Bool;
         INV_RESERVA2 : Bool;
      END_STRUCT;
      REFERENCIAS : Struct   // REFERÊNCIAS
         BASE : Real := 800.0;   // BASE DA MÁQUINA SEM ACC/DEC
         FINAL_MAQUINA : Real;   // FINAL DA MÁQUINA COM ACC/DEC
         TRABALHO : Real := 1005.0;   // TRABALHO DA MÁQUINA - 0=0M/MIN // 10.000=100M/MIN
         MINIMA : Real := 800.0;   // MINIMA DA MÁQUINA - 0=0M/MIN // 10.000=100M/MIN
         MAXIMA : Real := 8000.0;   // MAXIMA DA MÁQUINA - 0=0M/MIN // 10.000=100M/MIN
         PASSO_ACC : Real := 5.0;   // PASSO DE ACELERAÇÃO DA MÁQUINA
         PASSO_DEC : Real := 6.0;   // PASSO DE DESACELERAÇÃO DA MÁQUINA
         PASSO_DEC_NORMAL : Real := 6.0;   // PASSO DE DESACELERAÇÃO DA MÁQUINA - EM MARCHA
         PASSO_DEC_DESLIGA : Real := 9.0;   // PASSO DE DESACELERAÇÃO DA MÁQUINA - QUANDO A MÁQUINA ESTÁ DESLIGANDO
         PASSO_DEC_ALARME : Real := 25.0;   // PASSO DE DESACELERAÇÃO DA MÁQUINA - EM ALARME
      END_STRUCT;
      AUXILIARES1 : Struct
         HORIMETRO : Real := 183.0583;
         INVERSOR_RESERVA1 : Int;
         INVERSOR_RESERVA2 : Int;
      END_STRUCT;
   END_VAR
BEGIN
END_DATA_BLOCK

DATA_BLOCK "DB GRUPO 1"   // DB2
{ S7_Optimized_Access := 'FALSE' }
VERSION : 0.1
   VAR
      STAT0 : Struct
         STAT1 : Bool;
         STAT2 : Bool;
         STAT3 : Bool;
         STAT4 : Bool;
         STAT5 : Bool;
         STAT6 : Bool;
         STAT7 : Bool;
         STAT8 : Bool;
         STAT9 : Bool;
         STAT10 : Bool;
         STAT11 : Bool;
         STAT12 : Bool;
         STAT13 : Bool;
         STAT14 : Bool;
         STAT15 : Bool;
         STAT16 : Bool;
         STAT17 : Bool;
         STAT18 : Bool;
         STAT19 : Bool;
         STAT20 : Bool;
         STAT21 : Bool;
         STAT22 : Bool;
         STAT23 : Bool;
         STAT24 : Bool;
         STAT25 : Bool := TRUE;
         STAT26 : Bool;
         STAT27 : Bool;
         STAT28 : Bool;
         STAT29 : Bool;
         STAT30 : Bool;
         STAT31 : Bool;
         STAT32 : Bool;
         STAT33 : Bool;
         STAT34 : Bool;
         STAT35 : Bool;
         STAT36 : Bool;
         STAT37 : Bool;
         STAT38 : Bool;
         STAT39 : Bool;
         STAT40 : Bool;
         STAT41 : Bool;
         STAT42 : Bool;
         STAT43 : Bool;
         STAT44 : Bool;
         STAT45 : Bool;
         STAT46 : Bool;
         STAT47 : Word;
      END_STRUCT;
      STAT48 : Struct
         STAT49 : Bool := TRUE;
         STAT50 : Bool;
         STAT51 : Bool;
         STAT52 : Bool;
         STAT53 : Bool;
         STAT54 : Bool;
         STAT55 : Bool;
         STAT56 : Bool := TRUE;
         STAT57 : Bool;
         STAT58 : Bool;
         STAT59 : Bool;
         STAT60 : Bool;
         STAT61 : Bool;
         STAT62 : Bool;
         STAT63 : Bool;
         STAT64 : Bool;
         STAT65 : Bool;
         STAT66 : Bool;
         STAT67 : Bool;
         STAT68 : Bool;
         STAT69 : Bool;
         STAT70 : Bool := TRUE;
         STAT71 : Bool;
         STAT72 : Bool := TRUE;
         STAT73 : Bool;
         STAT74 : Bool;
         STAT75 : Bool;
         STAT76 : Bool;
         STAT77 : Bool;
         STAT78 : Bool;
         STAT79 : Bool;
         STAT80 : Bool;
         STAT81 : Bool;
         STAT82 : Bool;
         STAT83 : Bool;
         STAT84 : Bool;
         STAT85 : Bool;
         STAT86 : Bool;
         STAT87 : Bool;
         STAT88 : Bool;
         STAT89 : Bool;
         STAT90 : Bool;
         STAT91 : Bool;
         STAT92 : Bool;
         STAT93 : Bool;
         STAT94 : Bool;
         STAT95 : Bool;
      END_STRUCT;
      STAT96 : Struct
         STAT97 : Bool;
         STAT98 : Bool;
         STAT99 : Bool;
         STAT100 : Bool;
         STAT101 : Bool;
         STAT102 : Bool := TRUE;
         STAT103 : Bool;
         STAT104 : Bool;
         STAT105 : Bool;
         STAT106 : Bool := TRUE;
         STAT107 : Bool;
         STAT108 : Bool;
         STAT109 : Bool;
         STAT110 : Bool := TRUE;
         STAT111 : Bool;
         STAT112 : Bool;
         STAT113 : Bool;
         STAT114 : Bool;
         STAT115 : Bool;
         STAT116 : Bool;
         STAT117 : Bool;
         STAT118 : Bool;
         STAT119 : Bool;
         STAT120 : Bool;
         STAT121 : Bool;
         STAT122 : Bool;
         STAT123 : Bool;
         STAT124 : Bool;
         STAT125 : Bool;
         STAT126 : Bool;
         STAT127 : Bool := TRUE;
         STAT128 : Bool;
         STAT129 : Bool;
         STAT130 : Bool;
         STAT131 : Bool;
         STAT132 : Bool;
         STAT133 : Bool;
         STAT134 : Bool;
         STAT135 : Bool;
         STAT136 : Bool;
         STAT137 : Bool;
      END_STRUCT;
      STAT138 : Struct
         STAT139 : Real;
         STAT140 : Real;
         STAT141 : Real := 850.0;
         STAT142 : Real := 850.0;
         STAT143 : Real := 600.0;
         STAT144 : Real := 600.0;
         STAT145 : Real := 1500.0;
         STAT146 : Real := 750.0;
         STAT147 : Real := 750.0;
         STAT148 : Real := 750.0;
         STAT149 : Real := 750.0;
         STAT150 : Real;
         STAT151 : Real;
         STAT152 : Real;
         STAT153 : Real;
      END_STRUCT;
      STAT154 : Struct
         STAT155 : Real;
         STAT156 : Real;
         STAT157 : Real := 337.0;
         STAT158 : Real := 340.0;
         STAT159 : Real := 377.0;
         STAT160 : Real := 537.0;
         STAT161 : Real;
         STAT162 : Real := 359.0;
         STAT163 : Real := 358.0;
         STAT164 : Real := 357.0;
         STAT165 : Real := 369.0;
         STAT166 : Real := -16.59257;
      END_STRUCT;
   END_VAR
BEGIN
END_DATA_BLOCK

DATA_BLOCK "DB GRUPO 2"   // DB3
{ S7_Optimized_Access := 'FALSE' }
VERSION : 0.1
   VAR
      ALARMES : Struct
         TERM_ROSCA_FOULARD : Bool;
         TERM_EXAUSTOR_SECA1 : Bool;
         TERM_EXAUSTOR_SECA2 : Bool;
         TERM_EXAUSTOR_SECA3 : Bool;
         TERM_EXAUSTOR_SECA4 : Bool;
         ALAR_NIVEL_BAIXO_GOMA : Bool;   // ALARME DE NIVEL BAIXO CAIXA DE GOMA
         RESERVA2 : Word;
         RESERVA4 : Word;
         RESERVA6 : Word;
      END_STRUCT;
      COMANDO : Struct
         MAN_AUT_ROSCA_FOULARD : Bool := TRUE;
         LIG_DESL_ROSCA_FOULARD : Bool;
         LIG_EXAUSTOR_SECA1 : Bool;
         LIG_EXAUSTOR_SECA2 : Bool;
         LIG_EXAUSTOR_SECA3 : Bool;
         LIG_EXAUSTOR_SECA4 : Bool;
         LIG_NIVEL_FOULARD : Bool;
         RESERVA8_7 : Bool;
         LIG_DESL_TEMP_TQ1 : Bool := TRUE;
         RESERVA9_1 : Bool;
         LIG_DESL_TEMP_TQ2 : Bool := TRUE;
         RESERVA9_3 : Bool;
         LIG_DESL_TEMP_TQ3 : Bool;
         RESERVA9_5 : Bool;
         LIG_DESL_TEMP_TQ4 : Bool;
         RESERVA10 : Word;
         RESERVA12 : Word;
      END_STRUCT;
      STATUS : Struct
         ROSCA_FOULARD : Bool;
         EXAUSTOR_SECA1 : Bool;
         EXAUSTOR_SECA2 : Bool;
         EXAUSTOR_SECA3 : Bool;
         EXAUSTOR_SECA4 : Bool;
         NIVEL_FOULARD : Bool;
         VALVULA_PRODUTO_FOULARD : Bool;
         RESERVA14_7 : Bool;
         VALVULA_TQ1 : Bool;
         VALVULA_TQ2 : Bool;
         VALVULA_TQ3 : Bool;
         VALVULA_TQ4 : Bool;
         RESERVA16 : Word;
         RESERVA18 : Word;
      END_STRUCT;
      SETPOINT : Struct
         TEMP_TQ1 : Real := 400.0;
         TEMP_TQ2 : Real;
         TEMP_TQ3 : Real;
         TEMP_TQ4 : Real;
         RESERVA_36 : Real;
         RESERVA_40 : Real;
         RESERVA_44 : Real;
         RESERVA_48 : Real;
         RESERVA_52 : Real;
         RESERVA_56 : Real;
         RESERVA_60 : Real;
         RESERVA_64 : Real;
         RESERVA_68 : Real;
         RESERVA_72 : Real;
         RESERVA_76 : Real;
      END_STRUCT;
      VALOR_REAL : Struct
         TEMP_TQ1 : Real := 402.0;
         TEMP_TQ2 : Real := 323.0;
         TEMP_TQ3 : Real := 373.0;
         TEMP_TQ4 : Real := -32768.0;
         TEMP_FOULARD : Real := 280.0;
      END_STRUCT;
   END_VAR
BEGIN
END_DATA_BLOCK

DATA_BLOCK "DB PID"   // DB7
{ S7_Optimized_Access := 'FALSE' }
VERSION : 0.1
   VAR
      VALVULA_FLUXO1 : Word;
      VALVULA_FLUXO2 : Word;
      RESERVA_4 : Real;
      RESERVA_8 : Real;
      AUXILIAR : Struct
         NEUTRALIZACAO1 : Int;
         FLUXO_AGUA_CX1 : Int;
         FLUXO_AGUA_CX2 : Int;
         RESERVA_18 : Int;
         NEUTRALIZACAO2 : Int;
         RESERVA_22 : Int;
         RESERVA_24 : Int;
         RESERVA_26 : Int;
         SECADEIRA1 : Int;
         RESERVA_30 : Int;
         SECADEIRA2 : Int;
         SECADEIRA3 : Int;
         SECADEIRA4 : Int;
         RESERVA_38 : Int;
         RESERVA_40 : Int;
         RESERVA_42 : Int;
         RESERVA_44 : Int;
      END_STRUCT;
      SETPOINT : Struct
         NEUTRALIZACAO1 : Real := 850.0;
         FLUXO_AGUA_CX1 : Real;
         FLUXO_AGUA_CX2 : Real;
         RESERVA_52 : Real;
         NEUTRALIZACAO2 : Real;
         RESERVA_2 : Real;
         RESERVA_64 : Real;
         RESERVA_68 : Real;
         SECADEIRA1 : Real;
         RESERVA_3 : Real;
         SECADEIRA2 : Real := 1020.0;
         SECADEIRA3 : Real := 1070.0;
         SECADEIRA4 : Real := 1100.0;
         RESERVA_92 : Real;
         RESERVA_96 : Real;
         RESERVA_100 : Real;
         RESERVA_104 : Real;
      END_STRUCT;
      CONTROLE : Struct
         NEUTRALIZACAO1 : Bool;
         FLUXO_AGUA_CX1 : Bool;
         FLUXO_AGUA_CX2 : Bool;
         RESERVA114_3 : Bool;
         NEUTRALIZACAO2 : Bool;
         RESERVA114_5 : Bool;
         RESERVA114_6 : Bool;
         RESERVA114_7 : Bool;
         SECADEIRA1 : Bool;
         TEMP_UMIDADE : Bool := TRUE;
         SECADEIRA2 : Bool;
         SECADEIRA3 : Bool;
         SECADEIRA4 : Bool;
         RESERVA_116 : Word;
      END_STRUCT;
      VALVULA : Struct
         TROCADOR1 : Word;
         TROCADOR2 : Word;
         SECADEIRA1 : Word;
         SECADEIRA2 : Word;
         SECADEIRA3 : Word;
         SECADEIRA4 : Word;
      END_STRUCT;
      STATUS : Struct
         NEUTRALIZACAO1 : Bool;
         FLUXO_AGUA_CX1 : Bool;
         FLUXO_AGUA_CX2 : Bool;
         TANQUE2_LAVAGEM1 : Bool;
         NEUTRALIZACAO2 : Bool;
         RESERVA_2 : Bool;
         TANQUE1_LAVAGEM2 : Bool;
         TANQUE2_LAVAGEM2 : Bool;
         SECADEIRA1 : Bool;
         RESERVA_3 : Bool;
         SECADEIRA2 : Bool;
         SECADEIRA3 : Bool;
         SECADEIRA4 : Bool;
         RESERVA_132 : Word;
      END_STRUCT;
      VALOR_REAL : Struct
         NEUTRALIZACAO1 : Real := 921.0;
         NEUTRALIZACAO2 : Real := 280.0;
         SECADEIRA1 : Real := 622.0;
         SECADEIRA2 : Real := 676.0;
         SECADEIRA3 : Real := 404.0;
         SECADEIRA4 : Real := 760.0;
         FLUXO1 : Real := -32768.0;
         FLUXO2 : Real := -32768.0;
      END_STRUCT;
      UMIDADE : Struct
         SET_POINT : Real := 31.24997;
         VARIAVEL_DE_PROCESSO : Real := 12.87616;
         VARIAVEL_MANIPULADA : Word;
      END_STRUCT;
   END_VAR
BEGIN
END_DATA_BLOCK

DATA_BLOCK "DB PUXADOR"   // DB10
TITLE = Automation Pack Automação Indl. e Com. Ltda.
{ S7_Optimized_Access := 'FALSE' }
AUTHOR : THALLES
FAMILY : TRAÇÃO
NAME : SMT-15
VERSION : 0.1
// Cliente: Texima S/A Ind. de Máquinas
// Cliente Final: Cia. Fiação e Tecidos Santo Antonio.
// Máquina: Linha 1 DENIN - O.S.: 24.626
   VAR
      ALARMES : Struct   // ALARMES
         PROTECAO_INVERSOR : Bool;   // ALARME DE NIVEL ALTO - PROTEÇÃO DO INVERSOR DE FREQUENCIA
         PROTECAO_RESERVA : Bool;   // ALARME DE NIVEL ALTO - RESERVA
         BALANCA_INFERIOR : Bool;   // ALARME DE NIVEL ALTO - BALANÇA INFERIOR
         BALANCA_SUPERIOR : Bool;   // ALARME DE NIVEL ALTO - BALANÇA SUPERIOR
         RESERVA_10 : Byte;   // ALARME DE NIVEL ALTO - RESERVA
         RESERVA_20 : Byte;   // ALARME DE NIVEL BAIXO - RESERVA
         RESERVA_30 : Byte;   // ALARME DE NIVEL BAIXO - RESERVA
      END_STRUCT;
      COMANDOS : Struct   // COMANDOS
         SELECAO : Bool;   // COMANDO PARA SELEÇÃO "ON/OFF" - COMANDA O PROXIMO BIT...
         SELECIONADO : Bool;   // 1=MOTOR SELECIONADO
         JOG : Bool;   // 1= JOG
         MARCHA : Bool;   // 1=MARCHA
         FRENTE_REVERSAO : Bool;   // SENTIDO DE ROTAÇÃO DO MOTOR // 0=FRENTE - 1=REVERSÃO
         RESERVA_45 : Bool;   // RESERVA
         RESERVA_46 : Bool;   // RESERVA
         RESERVA_47 : Bool;   // RESERVA
         SINC_INDEP : Bool := TRUE;   // TIPO DE CONTROLE // 0=SINCRONIZADO - 1=INDEPENDENTE
         TROCA_ROLO : Bool;   // 1=MODO TROCA ROLO ATIVO
         CONTROLE_INDEPENDENTE : Bool;   // 1=CONTROLE INDEPENDENTE ATIVO
         SINCRONISMO_PUXADOR : Bool;   // AUXILIAR - REALIZA O SINCRONISMO DO PUXADOR COM A MÁQUINA APOS O TROCA ROLO
         JOG_SUPER : Bool;   // RESERVA
         RESERVA_55 : Bool;   // RESERVA
         RESERVA_56 : Bool;   // RESERVA
         RESERVA_57 : Bool;   // RESERVA
         RESERVA_60 : Byte;   // RESERVA
         RESERVA_70 : Bool;   // RESERVA
         RESERVA_71 : Bool;   // RESERVA
         RESERVA_72 : Bool;   // RESERVA
         RESERVA_73 : Bool;   // RESERVA
         RESERVA_74 : Bool;   // RESERVA
         RESERVA_75 : Bool;   // RESERVA
         STATUS_DRIVER : Bool := TRUE;   // BIT AUXILIAR DE STATUS DO INVERSOR DE FREQUENCIA - 1=OK
         DESBLOQUEIO_DRIVER : Bool;   // BIT AUXILIAR DE DESBLOQUEIO DO INVERSOR DE FREQÊNCIA
      END_STRUCT;
      REFERENCIAS : Struct   // REFERÊNCIAS
         BASE : Real;   // BASE SEM ACC/DEC
         FINAL : Real;   // FINAL COM ACC/DEC
         CORRECAO : Real;   // CORRECAO BALANCA
         BALANCA : Real := 80.46666;   // POSIÇÃO DA BALANÇA - -100...0...100%
         GANHO_BALANCA : Real;   // GANHO DA BALAÇA - 10%...30% - REFERENTE A VELOCIDADE MÁXIMA DA MÁQUINA
         INDEPENDENTE : Real;   // REFERÊNCIA INDEPENDENTE - AJUSTADA PELO POTENCIÔMETRO NA REMOTA DO PUXADOR
         RESERVA_320 : Real;   // RESERVA
         RESERVA_360 : Real;   // RESERVA
         RESERVA_400 : Real;   // RESERVA
         RESERVA_440 : Real;   // RESERVA
         VELOCIDADE_MAXIMA : Real := 8000.0;   // VELOCIDADE MAXIMA - 0=0M/MIN // 10.000=100M/MIN - CALCULADO AUTOMÁTICAMENTE
      END_STRUCT;
      RESERVA_520 : Byte;   // RESERVA
      RESERVA_530 : Byte;   // RESERVA
      RESERVA_540 : Byte;   // RESERVA
      RESERVA_550 : Byte;   // RESERVA
      RESERVA_560 : Byte;   // RESERVA
      RESERVA_570 : Byte;   // RESERVA
      RESERVA_580 : Byte;   // RESERVA
      RESERVA_590 : Byte;   // RESERVA
   END_VAR
BEGIN
END_DATA_BLOCK

DATA_BLOCK "DB CHAMUSCADEIRA"   // DB11
TITLE = Automation Pack Automação Indl. e Com. Ltda.
{ S7_Optimized_Access := 'FALSE' }
AUTHOR : THALLES
FAMILY : TRAÇÃO
NAME : LINHA1
VERSION : 0.1
// Cliente: Texima S/A Ind. de Máquinas
// Cliente Final: Cia. Fiação e Tecidos Santo Antonio.
// Máquina: Linha 1 DENIN - O.S.: 24.626
   VAR
      ALARMES : Struct   // ALARMES
         PROTECAO_INVERSOR : Bool;   // ALARME DE NIVEL ALTO - PROTEÇÃO DO INVERSOR DE FREQUENCIA
         RESERVA_01 : Bool;   // ALARME DE NIVEL ALTO - RESERVA
         BALANCA_INFERIOR : Bool;   // ALARME DE NIVEL ALTO - BALANÇA INFERIOR
         BALANCA_SUPERIOR : Bool;   // ALARME DE NIVEL ALTO - BALANÇA SUPERIOR
         RESERVA_10 : Byte;   // ALARME DE NIVEL ALTO - RESERVA
         RESERVA_20 : Byte;   // ALARME DE NIVEL BAIXO - RESERVA
         RESERVA_30 : Byte;   // ALARME DE NIVEL BAIXO - RESERVA
      END_STRUCT;
      COMANDOS : Struct   // COMANDOS
         SELECAO : Bool;   // COMANDO PARA SELEÇÃO "ON/OFF" - COMANDA O PROXIMO BIT...
         SELECIONADO : Bool;   // 1=MOTOR SELECIONADO
         JOG : Bool;   // 1=JOG
         MARCHA : Bool;   // 1=MARCHA
         FRENTE_REVERSAO : Bool;   // SENTIDO DE ROTAÇÃO DO MOTOR // 0=FRENTE - 1=REVERSÃO
         RESERVA_5 : Byte;   // RESERVA
         RESERVA_6 : Byte;   // RESERVA
         RESERVA_30 : Bool;   // RESERVA
         RESERVA_31 : Bool;   // RESERVA
         RESERVA_32 : Bool;   // RESERVA
         RESERVA_33 : Bool;   // RESERVA
         RESERVA_34 : Bool;   // RESERVA
         RESERVA_35 : Bool;   // RESERVA
         STATUS_DRIVER : Bool := TRUE;   // BIT AUXILIAR DE STATUS DO INVERSOR DE FREQUENCIA - 1=OK
         DESBLOQUEIO_DRIVER : Bool;   // BIT AUXILIAR DE DESBLOQUEIO DO INVERSOR DE FREQÊNCIA
      END_STRUCT;
      REFERENCIAS : Struct   // REFERÊNCIAS
         BASE : Real;   // BASE SEM ACC/DEC
         FINAL : Real;   // FINAL COM ACC/DEC
         CORRECAO : Real;   // CORRECAO BALANCA
         BALANCA : Real := -100.0;   // POSIÇÃO DA BALANÇA - -100...0...100%
         GANHO_BALANCA : Real;   // GANHO DA BALAÇA - 10%...30% - REFERENTE A VELOCIDADE MÁXIMA DA MÁQUINA
         RESERVA_28 : Real;   // RESERVA
         RESERVA_32 : Real;   // RESERVA
         RESERVA_36 : Real;   // RESERVA
         RESERVA_40 : Real;   // RESERVA
         RESERVA_44 : Real;   // RESERVA
         VELOCIDADE_MAXIMA : Real := 8000.0;   // VELOCIDADE MAXIMA - 0=0M/MIN // 10.000=100M/MIN - CALCULADO AUTOMÁTICAMENTE
      END_STRUCT;
   END_VAR
BEGIN
END_DATA_BLOCK

DATA_BLOCK "DB NEUTRALIZACAO1"   // DB12
TITLE = Automation Pack Automação Indl. e Com. Ltda.
{ S7_Optimized_Access := 'FALSE' }
AUTHOR : THALLES
FAMILY : TRAÇÃO
NAME : LINHA1
VERSION : 0.1
// Cliente: Texima S/A Ind. de Máquinas
// Cliente Final: Cia. Fiação e Tecidos Santo Antonio.
// Máquina: Linha 1 DENIN - O.S.: 24.626
   VAR
      ALARMES : Struct   // ALARMES
         PROTECAO_INVERSOR : Bool;   // ALARME DE NIVEL ALTO - PROTEÇÃO DO INVERSOR DE FREQUENCIA
         RESERVA_01 : Bool;   // ALARME DE NIVEL ALTO - RESERVA
         BALANCA_INFERIOR : Bool;   // ALARME DE NIVEL ALTO - BALANÇA INFERIOR
         BALANCA_SUPERIOR : Bool;   // ALARME DE NIVEL ALTO - BALANÇA SUPERIOR
         RESERVA_1 : Byte;   // ALARME DE NIVEL ALTO - RESERVA
         RESERVA_2 : Byte;   // ALARME DE NIVEL BAIXO - RESERVA
         RESERVA_3 : Byte;   // ALARME DE NIVEL BAIXO - RESERVA
      END_STRUCT;
      COMANDOS : Struct   // COMANDOS
         SELECAO : Bool;   // COMANDO PARA SELEÇÃO "ON/OFF" - COMANDA O PROXIMO BIT...
         SELECIONADO : Bool;   // 1=MOTOR SELECIONADO
         JOG : Bool;   // 1=JOG
         MARCHA : Bool;   // 1=MARCHA
         FRENTE_REVERSAO : Bool;   // SENTIDO DE ROTAÇÃO DO MOTOR // 0=FRENTE - 1=REVERSÃO
         RESERVA_05 : Bool;   // RESERVA
         TAXA_BALANCA : Bool;   // TIPO DE CONTROLE // 0=TAXA - 1=BALANÇA
         ACAO_BALANCA : Bool;   // AÇÃO DA BALANÇA // 0=DIRETA - 1=REVERSA
         RESERVA_5 : Byte;   // RESERVA
         RESERVA_6 : Byte;   // RESERVA
         RESERVA_30 : Bool;   // RESERVA
         RESERVA_31 : Bool;   // RESERVA
         RESERVA_32 : Bool;   // RESERVA
         RESERVA_33 : Bool;   // RESERVA
         RESERVA_34 : Bool;   // RESERVA
         RESERVA_35 : Bool;   // RESERVA
         STATUS_DRIVER : Bool := TRUE;   // BIT AUXILIAR DE STATUS DO INVERSOR DE FREQUENCIA - 1=OK
         DESBLOQUEIO_DRIVER : Bool;   // BIT AUXILIAR DE DESBLOQUEIO DO INVERSOR DE FREQÊNCIA
      END_STRUCT;
      REFERENCIAS : Struct   // REFERÊNCIAS
         BASE : Real;   // BASE SEM ACC/DEC
         FINAL : Real;   // FINAL COM ACC/DEC
         CORRECAO : Real;   // CORRECAO BALANCA
         BALANCA : Real := 100.0;   // POSIÇÃO DA BALANÇA - -100...0...100%
         GANHO_BALANCA : Real;   // GANHO DA BALAÇA - 10%...30% - REFERENTE A VELOCIDADE MÁXIMA DA MÁQUINA
         RESERVA_28 : Real;   // RESERVA
         RESERVA_32 : Real;   // RESERVA
         RESERVA_36 : Real;   // RESERVA
         RESERVA_40 : Real;   // RESERVA
         RESERVA_44 : Real;   // RESERVA
         VELOCIDADE_MAXIMA : Real := 8000.0;   // VELOCIDADE MAXIMA - 0=0M/MIN // 10.000=100M/MIN - CALCULADO AUTOMÁTICAMENTE
      END_STRUCT;
   END_VAR
BEGIN
END_DATA_BLOCK

DATA_BLOCK "DB EXTRACTA1"   // DB13
TITLE = Automation Pack Automação Indl. e Com. Ltda.
{ S7_Optimized_Access := 'FALSE' }
AUTHOR : THALLES
FAMILY : TRAÇÃO
NAME : LINHA1
VERSION : 0.1
// Cliente: Texima S/A Ind. de Máquinas
// Cliente Final: Cia. Fiação e Tecidos Santo Antonio.
// Máquina: Linha 1 DENIN - O.S.: 24.626
   VAR
      STAT0 : Struct
         STAT1 : Bool;
         STAT2 : Bool;
         STAT3 : Byte;
         STAT4 : Byte;
         STAT5 : Byte;
      END_STRUCT;
      STAT6 : Struct
         STAT7 : Bool;
         STAT8 : Bool;
         STAT9 : Bool;
         STAT10 : Bool;
         STAT11 : Bool;
         STAT12 : Bool;
         STAT13 : Bool;
         STAT14 : Byte;
         STAT15 : Byte;
         STAT16 : Bool;
         STAT17 : Bool;
         STAT18 : Bool;
         STAT19 : Bool;
         STAT20 : Bool;
         STAT21 : Bool;
         STAT22 : Bool := TRUE;
         STAT23 : Bool;
      END_STRUCT;
      STAT24 : Struct
         STAT25 : Real;
         STAT26 : Real;
         STAT27 : Real := -3244.444;
         STAT28 : Real;
         STAT29 : Real;
         STAT30 : Real := 9600.0;
         STAT31 : Real;
         STAT32 : Real;
         STAT33 : Real;
         STAT34 : Real;
         STAT35 : Real := 9600.0;
      END_STRUCT;
   END_VAR
BEGIN
END_DATA_BLOCK

DATA_BLOCK "DB LAVAGEM1"   // DB14
TITLE = Automation Pack Automação Indl. e Com. Ltda.
{ S7_Optimized_Access := 'FALSE' }
AUTHOR : THALLES
FAMILY : TRAÇÃO
NAME : LINHA1
VERSION : 0.1
// Cliente: Texima S/A Ind. de Máquinas
// Cliente Final: Cia. Fiação e Tecidos Santo Antonio.
// Máquina: Linha 1 DENIN - O.S.: 24.626
   VAR
      ALARMES : Struct   // ALARMES
         PROTECAO_INVERSOR : Bool;   // ALARME DE NIVEL ALTO - PROTEÇÃO DO INVERSOR DE FREQUENCIA
         RESERVA_01 : Bool;   // ALARME DE NIVEL ALTO - RESERVA
         BALANCA_INFERIOR : Bool;   // ALARME DE NIVEL ALTO - BALANÇA INFERIOR
         BALANCA_SUPERIOR : Bool;   // ALARME DE NIVEL ALTO - BALANÇA SUPERIOR
         RESERVA_10 : Byte;   // ALARME DE NIVEL ALTO - RESERVA
         RESERVA_20 : Byte;   // ALARME DE NIVEL BAIXO - RESERVA
         RESERVA_30 : Byte;   // ALARME DE NIVEL BAIXO - RESERVA
      END_STRUCT;
      COMANDOS : Struct   // COMANDOS
         SELECAO : Bool;   // COMANDO PARA SELEÇÃO "ON/OFF" - COMANDA O PROXIMO BIT...
         SELECIONADO : Bool;   // 1=MOTOR SELECIONADO
         JOG : Bool;   // 1=JOG
         MARCHA : Bool;   // 1=MARCHA
         FRENTE_REVERSAO : Bool;   // SENTIDO DE ROTAÇÃO DO MOTOR // 0=FRENTE - 1=REVERSÃO
         RESERVA_5 : Byte;   // RESERVA
         RESERVA_6 : Byte;   // RESERVA
         RESERVA_30 : Bool;   // RESERVA
         RESERVA_31 : Bool;   // RESERVA
         RESERVA_32 : Bool;   // RESERVA
         RESERVA_33 : Bool;   // RESERVA
         RESERVA_34 : Bool;   // RESERVA
         RESERVA_35 : Bool;   // RESERVA
         STATUS_DRIVER : Bool := TRUE;   // BIT AUXILIAR DE STATUS DO INVERSOR DE FREQUENCIA - 1=OK
         DESBLOQUEIO_DRIVER : Bool;   // BIT AUXILIAR DE DESBLOQUEIO DO INVERSOR DE FREQÊNCIA
      END_STRUCT;
      REFERENCIAS : Struct   // REFERÊNCIAS
         BASE : Real;   // BASE SEM ACC/DEC
         FINAL : Real;   // FINAL COM ACC/DEC
         CORRECAO : Real;   // CORRECAO BALANCA
         BALANCA : Real := 61.94452;   // POSIÇÃO DA BALANÇA - -100...0...100%
         GANHO_BALANCA : Real;   // GANHO DA BALAÇA - 10%...30% - REFERENTE A VELOCIDADE MÁXIMA DA MÁQUINA
         RESERVA_28 : Real;   // RESERVA
         RESERVA_32 : Real;   // RESERVA
         RESERVA_36 : Real;   // RESERVA
         RESERVA_40 : Real;   // RESERVA
         RESERVA_44 : Real;   // RESERVA
         VELOCIDADE_MAXIMA : Real := 8000.0;   // VELOCIDADE MAXIMA - 0=0M/MIN // 10.000=100M/MIN - CALCULADO AUTOMÁTICAMENTE
      END_STRUCT;
   END_VAR
BEGIN
END_DATA_BLOCK

DATA_BLOCK "DB NEUTRALIZACAO2"   // DB15
TITLE = Automation Pack Automação Indl. e Com. Ltda.
{ S7_Optimized_Access := 'FALSE' }
AUTHOR : THALLES
FAMILY : TRAÇÃO
NAME : LINHA1
VERSION : 0.1
// Cliente: Texima S/A Ind. de Máquinas
// Cliente Final: Cia. Fiação e Tecidos Santo Antonio.
// Máquina: Linha 1 DENIN - O.S.: 24.626
   VAR
      ALARMES : Struct   // ALARMES
         PROTECAO_INVERSOR : Bool;   // ALARME DE NIVEL ALTO - PROTEÇÃO DO INVERSOR DE FREQUENCIA
         RESERVA_01 : Bool;   // ALARME DE NIVEL ALTO - RESERVA
         BALANCA_INFERIOR : Bool;   // ALARME DE NIVEL ALTO - BALANÇA INFERIOR
         BALANCA_SUPERIOR : Bool;   // ALARME DE NIVEL ALTO - BALANÇA SUPERIOR
         RESERVA_10 : Byte;   // ALARME DE NIVEL ALTO - RESERVA
         RESERVA_20 : Byte;   // ALARME DE NIVEL BAIXO - RESERVA
         RESERVA_30 : Byte;   // ALARME DE NIVEL BAIXO - RESERVA
      END_STRUCT;
      COMANDOS : Struct   // COMANDOS
         SELECAO : Bool;   // COMANDO PARA SELEÇÃO "ON/OFF" - COMANDA O PROXIMO BIT...
         SELECIONADO : Bool;   // 1=MOTOR SELECIONADO
         JOG : Bool;   // 1=JOG
         MARCHA : Bool;   // 1=MARCHA
         FRENTE_REVERSAO : Bool;   // SENTIDO DE ROTAÇÃO DO MOTOR // 0=FRENTE - 1=REVERSÃO
         RESERVA_5 : Byte;   // RESERVA
         RESERVA_6 : Byte;   // RESERVA
         RESERVA_30 : Bool;   // RESERVA
         RESERVA_31 : Bool;   // RESERVA
         RESERVA_32 : Bool;   // RESERVA
         RESERVA_33 : Bool;   // RESERVA
         RESERVA_34 : Bool;   // RESERVA
         RESERVA_35 : Bool;   // RESERVA
         STATUS_DRIVER : Bool := TRUE;   // BIT AUXILIAR DE STATUS DO INVERSOR DE FREQUENCIA - 1=OK
         DESBLOQUEIO_DRIVER : Bool;   // BIT AUXILIAR DE DESBLOQUEIO DO INVERSOR DE FREQÊNCIA
      END_STRUCT;
      REFERENCIAS : Struct   // REFERÊNCIAS
         BASE : Real;   // BASE SEM ACC/DEC
         FINAL : Real;   // FINAL COM ACC/DEC
         CORRECAO : Real;   // CORRECAO BALANCA
         BALANCA : Real := -100.0;   // POSIÇÃO DA BALANÇA - -100...0...100%
         GANHO_BALANCA : Real;   // GANHO DA BALAÇA - 10%...30% - REFERENTE A VELOCIDADE MÁXIMA DA MÁQUINA
         RESERVA_28 : Real;   // RESERVA
         RESERVA_32 : Real;   // RESERVA
         RESERVA_36 : Real;   // RESERVA
         RESERVA_40 : Real;   // RESERVA
         RESERVA_44 : Real;   // RESERVA
         VELOCIDADE_MAXIMA : Real := 8384.0;   // VELOCIDADE MAXIMA - 0=0M/MIN // 10.000=100M/MIN - CALCULADO AUTOMÁTICAMENTE
      END_STRUCT;
   END_VAR
BEGIN
END_DATA_BLOCK

DATA_BLOCK "DB EXTRACTA2"   // DB16
TITLE = Automation Pack Automação Indl. e Com. Ltda.
{ S7_Optimized_Access := 'FALSE' }
AUTHOR : THALLES
FAMILY : TRAÇÃO
NAME : LINHA1
VERSION : 0.1
// Cliente: Texima S/A Ind. de Máquinas
// Cliente Final: Cia. Fiação e Tecidos Santo Antonio.
// Máquina: Linha 1 DENIN - O.S.: 24.626
   VAR
      ALARMES : Struct   // ALARMES
         PROTECAO_INVERSOR : Bool;   // ALARME DE NIVEL ALTO - PROTEÇÃO DO INVERSOR DE FREQUENCIA
         Celula : Bool;   // Celula de carga trabalhando acima do maximo
         RESERVA_10 : Byte;   // ALARME DE NIVEL ALTO - RESERVA
         RESERVA_20 : Byte;   // ALARME DE NIVEL BAIXO - RESERVA
         RESERVA_30 : Byte;   // ALARME DE NIVEL BAIXO - RESERVA
      END_STRUCT;
      COMANDOS : Struct   // COMANDOS
         SELECAO : Bool;   // COMANDO PARA SELEÇÃO "ON/OFF" - COMANDA O PROXIMO BIT...
         SELECIONADO : Bool;   // 1=MOTOR SELECIONADO
         JOG : Bool;   // 1=JOG
         MARCHA : Bool;   // 1=MARCHA
         FRENTE_REVERSAO : Bool;   // SENTIDO DE ROTAÇÃO DO MOTOR // 0=FRENTE - 1=REVERSÃO
         RESERVA_5 : Byte;   // RESERVA
         RESERVA_6 : Byte;   // RESERVA
         RESERVA_30 : Bool;   // RESERVA
         RESERVA_31 : Bool;   // RESERVA
         RESERVA_32 : Bool;   // RESERVA
         RESERVA_33 : Bool;   // RESERVA
         RESERVA_34 : Bool;   // RESERVA
         RESERVA_35 : Bool;   // RESERVA
         STATUS_DRIVER : Bool := TRUE;   // BIT AUXILIAR DE STATUS DO INVERSOR DE FREQUENCIA - 1=OK
         DESBLOQUEIO_DRIVER : Bool;   // BIT AUXILIAR DE DESBLOQUEIO DO INVERSOR DE FREQÊNCIA
      END_STRUCT;
      REFERENCIAS : Struct   // REFERÊNCIAS
         BASE : Real;   // BASE SEM ACC/DEC
         FINAL : Real;   // FINAL COM ACC/DEC
         CORRECAO : Real := -1348.148;   // CORRECAO DA CELULA DE CARGA
         CELULA_REAL : Real;   // VALOR REAL DA CELULA DE CARGA
         RESERVA_24 : Real;   // RESERVA
         RESERVA_28 : Real := 9600.0;   // RESERVA
         RESERVA_32 : Real;   // RESERVA
         RESERVA_36 : Real;   // RESERVA
         RESERVA_40 : Real;   // RESERVA
         RESERVA_44 : Real;   // RESERVA
         VELOCIDADE_MAXIMA : Real := 9600.0;   // VELOCIDADE MAXIMA - 0=0M/MIN // 10.000=100M/MIN - CALCULADO AUTOMÁTICAMENTE
      END_STRUCT;
   END_VAR
BEGIN
END_DATA_BLOCK

DATA_BLOCK "DB LAVAGEM2"   // DB17
TITLE = Automation Pack Automação Indl. e Com. Ltda.
{ S7_Optimized_Access := 'FALSE' }
AUTHOR : THALLES
FAMILY : TRAÇÃO
NAME : LINHA1
VERSION : 0.1
// Cliente: Texima S/A Ind. de Máquinas
// Cliente Final: Cia. Fiação e Tecidos Santo Antonio.
// Máquina: Linha 1 DENIN - O.S.: 24.626
   VAR
      ALARMES : Struct   // ALARMES
         PROTECAO_INVERSOR : Bool;   // ALARME DE NIVEL ALTO - PROTEÇÃO DO INVERSOR DE FREQUENCIA
         RESERVA_01 : Bool;   // ALARME DE NIVEL ALTO - RESERVA
         BALANCA_INFERIOR : Bool;   // ALARME DE NIVEL ALTO - BALANÇA INFERIOR
         BALANCA_SUPERIOR : Bool;   // ALARME DE NIVEL ALTO - BALANÇA SUPERIOR
         RESERVA_10 : Byte;   // ALARME DE NIVEL ALTO - RESERVA
         RESERVA_20 : Byte;   // ALARME DE NIVEL BAIXO - RESERVA
         RESERVA_30 : Byte;   // ALARME DE NIVEL BAIXO - RESERVA
      END_STRUCT;
      COMANDOS : Struct   // COMANDOS
         SELECAO : Bool;   // COMANDO PARA SELEÇÃO "ON/OFF" - COMANDA O PROXIMO BIT...
         SELECIONADO : Bool;   // 1=MOTOR SELECIONADO
         JOG : Bool;   // 1=JOG
         MARCHA : Bool;   // 1=MARCHA
         FRENTE_REVERSAO : Bool;   // SENTIDO DE ROTAÇÃO DO MOTOR // 0=FRENTE - 1=REVERSÃO
         RESERVA_5 : Byte;   // RESERVA
         RESERVA_6 : Byte;   // RESERVA
         RESERVA_30 : Bool;   // RESERVA
         RESERVA_31 : Bool;   // RESERVA
         RESERVA_32 : Bool;   // RESERVA
         RESERVA_33 : Bool;   // RESERVA
         RESERVA_34 : Bool;   // RESERVA
         RESERVA_35 : Bool;   // RESERVA
         STATUS_DRIVER : Bool := TRUE;   // BIT AUXILIAR DE STATUS DO INVERSOR DE FREQUENCIA - 1=OK
         DESBLOQUEIO_DRIVER : Bool;   // BIT AUXILIAR DE DESBLOQUEIO DO INVERSOR DE FREQÊNCIA
      END_STRUCT;
      REFERENCIAS : Struct   // REFERÊNCIAS
         BASE : Real;   // BASE SEM ACC/DEC
         FINAL : Real;   // FINAL COM ACC/DEC
         CORRECAO : Real;   // CORRECAO BALANCA
         BALANCA : Real := 100.0;   // POSIÇÃO DA BALANÇA - -100...0...100%
         GANHO_BALANCA : Real;   // GANHO DA BALAÇA - 10%...30% - REFERENTE A VELOCIDADE MÁXIMA DA MÁQUINA
         RESERVA_28 : Real;   // RESERVA
         RESERVA_32 : Real;   // RESERVA
         RESERVA_36 : Real;   // RESERVA
         RESERVA_40 : Real;   // RESERVA
         RESERVA_44 : Real;   // RESERVA
         VELOCIDADE_MAXIMA : Real := 8000.0;   // VELOCIDADE MAXIMA - 0=0M/MIN // 10.000=100M/MIN - CALCULADO AUTOMÁTICAMENTE
      END_STRUCT;
   END_VAR
BEGIN
END_DATA_BLOCK

DATA_BLOCK "DB SECADEIRA1"   // DB18
TITLE = Automation Pack Automação Indl. e Com. Ltda.
{ S7_Optimized_Access := 'FALSE' }
AUTHOR : THALLES
FAMILY : TRAÇÃO
NAME : LINHA1
VERSION : 0.1
// Cliente: Texima S/A Ind. de Máquinas
// Cliente Final: Cia. Fiação e Tecidos Santo Antonio.
// Máquina: Linha 1 DENIN - O.S.: 24.626
   VAR
      ALARMES : Struct   // ALARMES
         PROTECAO_INVERSOR : Bool;   // ALARME DE NIVEL ALTO - PROTEÇÃO DO INVERSOR DE FREQUENCIA
         RESERVA_01 : Bool;   // ALARME DE NIVEL ALTO - RESERVA
         BALANCA_INFERIOR : Bool;   // ALARME DE NIVEL ALTO - BALANÇA INFERIOR
         BALANCA_SUPERIOR : Bool;   // ALARME DE NIVEL ALTO - BALANÇA SUPERIOR
         RESERVA_10 : Byte;   // ALARME DE NIVEL ALTO - RESERVA
         RESERVA_20 : Byte;   // ALARME DE NIVEL BAIXO - RESERVA
         RESERVA_30 : Byte;   // ALARME DE NIVEL BAIXO - RESERVA
      END_STRUCT;
      COMANDOS : Struct   // COMANDOS
         SELECAO : Bool;   // COMANDO PARA SELEÇÃO "ON/OFF" - COMANDA O PROXIMO BIT...
         SELECIONADO : Bool;   // 1=MOTOR SELECIONADO
         JOG : Bool;   // 1=JOG
         MARCHA : Bool;   // 1=MARCHA
         FRENTE_REVERSAO : Bool;   // SENTIDO DE ROTAÇÃO DO MOTOR // 0=FRENTE - 1=REVERSÃO
         RESERVA_5 : Byte;   // RESERVA
         RESERVA_6 : Byte;   // RESERVA
         RESERVA_30 : Bool;   // RESERVA
         RESERVA_31 : Bool;   // RESERVA
         RESERVA_32 : Bool;   // RESERVA
         RESERVA_33 : Bool;   // RESERVA
         RESERVA_34 : Bool;   // RESERVA
         RESERVA_35 : Bool;   // RESERVA
         STATUS_DRIVER : Bool := TRUE;   // BIT AUXILIAR DE STATUS DO INVERSOR DE FREQUENCIA - 1=OK
         DESBLOQUEIO_DRIVER : Bool;   // BIT AUXILIAR DE DESBLOQUEIO DO INVERSOR DE FREQÊNCIA
      END_STRUCT;
      REFERENCIAS : Struct   // REFERÊNCIAS
         BASE : Real;   // BASE SEM ACC/DEC
         FINAL : Real;   // FINAL COM ACC/DEC
         CORRECAO : Real;   // CORRECAO BALANCA
         BALANCA : Real := -100.0;   // POSIÇÃO DA BALANÇA - -100...0...100%
         GANHO_BALANCA : Real;   // GANHO DA BALAÇA - 10%...30% - REFERENTE A VELOCIDADE MÁXIMA DA MÁQUINA
         RESERVA_28 : Real;   // RESERVA
         RESERVA_32 : Real;   // RESERVA
         RESERVA_36 : Real;   // RESERVA
         RESERVA_40 : Real;   // RESERVA
         RESERVA_44 : Real;   // RESERVA
         VELOCIDADE_MAXIMA : Real := 8000.0;   // VELOCIDADE MAXIMA - 0=0M/MIN // 10.000=100M/MIN - CALCULADO AUTOMÁTICAMENTE
      END_STRUCT;
   END_VAR
BEGIN
END_DATA_BLOCK

DATA_BLOCK "DB FOULARD"   // DB19
TITLE = Automation Pack Automação Indl. e Com. Ltda.
{ S7_Optimized_Access := 'FALSE' }
AUTHOR : THALLES
FAMILY : TRAÇÃO
NAME : LINHA1
VERSION : 0.1
// Cliente: Texima S/A Ind. de Máquinas
// Cliente Final: Cia. Fiação e Tecidos Santo Antonio.
// Máquina: Linha 1 DENIN - O.S.: 24.626
   VAR
      STAT0 : Struct
         STAT1 : Bool;
         STAT2 : Byte;
         STAT3 : Byte;
         STAT4 : Byte;
      END_STRUCT;
      STAT5 : Struct
         STAT6 : Bool;
         STAT7 : Bool;
         STAT8 : Bool;
         STAT9 : Bool;
         STAT10 : Bool;
         STAT11 : Byte;
         STAT12 : Byte;
         STAT13 : Bool;
         STAT14 : Bool;
         STAT15 : Bool;
         STAT16 : Bool;
         STAT17 : Bool;
         STAT18 : Bool;
         STAT19 : Bool := TRUE;
         STAT20 : Bool;
      END_STRUCT;
      STAT21 : Struct
         STAT22 : Real;
         STAT23 : Real;
         STAT24 : Real;
         STAT25 : Real;
         STAT26 : Real;
         STAT27 : Real;
         STAT28 : Real;
         STAT29 : Real;
         STAT30 : Real;
         STAT31 : Real;
         STAT32 : Real := 8000.0;
      END_STRUCT;
   END_VAR
BEGIN
END_DATA_BLOCK

DATA_BLOCK "DB ESTICADOR"   // DB20
TITLE = Automation Pack Automação Indl. e Com. Ltda.
{ S7_Optimized_Access := 'FALSE' }
AUTHOR : THALLES
FAMILY : TRAÇÃO
NAME : LINHA1
VERSION : 0.1
// Cliente: Texima S/A Ind. de Máquinas
// Cliente Final: Cia. Fiação e Tecidos Santo Antonio.
// Máquina: Linha 1 DENIN - O.S.: 24.626
   VAR
      ALARMES : Struct   // ALARMES
         PROTECAO_INVERSOR : Bool;   // ALARME DE NIVEL ALTO - PROTEÇÃO DO INVERSOR DE FREQUENCIA
         RESERVA_01 : Bool;   // ALARME DE NIVEL ALTO - RESERVA
         BALANCA_INFERIOR : Bool;   // ALARME DE NIVEL ALTO - BALANÇA INFERIOR
         BALANCA_SUPERIOR : Bool;   // ALARME DE NIVEL ALTO - BALANÇA SUPERIOR
         RESERVA_10 : Byte;   // ALARME DE NIVEL ALTO - RESERVA
         RESERVA_20 : Byte;   // ALARME DE NIVEL BAIXO - RESERVA
         RESERVA_30 : Byte;   // ALARME DE NIVEL BAIXO - RESERVA
      END_STRUCT;
      COMANDOS : Struct   // COMANDOS
         SELECAO : Bool;   // COMANDO PARA SELEÇÃO "ON/OFF" - COMANDA O PROXIMO BIT...
         SELECIONADO : Bool := TRUE;   // 1=MOTOR SELECIONADO
         JOG : Bool;   // 1=JOG
         MARCHA : Bool;   // 1=MARCHA
         FRENTE_REVERSAO : Bool;   // SENTIDO DE ROTAÇÃO DO MOTOR // 0=FRENTE - 1=REVERSÃO
         RESERVA_5 : Byte;   // RESERVA
         RESERVA_6 : Byte;   // RESERVA
         RESERVA_30 : Bool;   // RESERVA
         RESERVA_31 : Bool;   // RESERVA
         RESERVA_32 : Bool;   // RESERVA
         RESERVA_33 : Bool;   // RESERVA
         RESERVA_34 : Bool;   // RESERVA
         RESERVA_35 : Bool;   // RESERVA
         STATUS_DRIVER : Bool := TRUE;   // BIT AUXILIAR DE STATUS DO INVERSOR DE FREQUENCIA - 1=OK
         DESBLOQUEIO_DRIVER : Bool;   // BIT AUXILIAR DE DESBLOQUEIO DO INVERSOR DE FREQÊNCIA
      END_STRUCT;
      REFERENCIAS : Struct   // REFERÊNCIAS
         BASE : Real;   // BASE SEM ACC/DEC
         FINAL : Real;   // FINAL COM ACC/DEC
         CORRECAO : Real;   // CORRECAO BALANCA
         BALANCA : Real := 10.58823;   // POSIÇÃO DA BALANÇA - -100...0...100%
         GANHO_BALANCA : Real;   // GANHO DA BALAÇA - 10%...30% - REFERENTE A VELOCIDADE MÁXIMA DA MÁQUINA
         RESERVA_28 : Real;   // RESERVA
         RESERVA_32 : Real;   // RESERVA
         RESERVA_36 : Real;   // RESERVA
         RESERVA_40 : Real;   // RESERVA
         RESERVA_44 : Real;   // RESERVA
         VELOCIDADE_MAXIMA : Real := 8000.0;   // VELOCIDADE MAXIMA - 0=0M/MIN // 10.000=100M/MIN - CALCULADO AUTOMÁTICAMENTE
      END_STRUCT;
   END_VAR
BEGIN
END_DATA_BLOCK

DATA_BLOCK "DB PUXADOR_SECADEIRA2"   // DB21
TITLE = Automation Pack Automação Indl. e Com. Ltda.
{ S7_Optimized_Access := 'FALSE' }
AUTHOR : THALLES
FAMILY : TRAÇÃO
NAME : LINHA1
VERSION : 0.1
// Cliente: Texima S/A Ind. de Máquinas
// Cliente Final: Cia. Fiação e Tecidos Santo Antonio.
// Máquina: Linha 1 DENIN - O.S.: 24.626
   VAR
      ALARMES : Struct   // ALARMES
         PROTECAO_INVERSOR : Bool;   // ALARME DE NIVEL ALTO - PROTEÇÃO DO INVERSOR DE FREQUENCIA
         RESERVA_1 : Byte;   // ALARME DE NIVEL ALTO - RESERVA
         RESERVA_2 : Byte;   // ALARME DE NIVEL BAIXO - RESERVA
         RESERVA_3 : Byte;   // ALARME DE NIVEL BAIXO - RESERVA
      END_STRUCT;
      COMANDOS : Struct   // COMANDOS
         SELECAO : Bool;   // COMANDO PARA SELEÇÃO "ON/OFF" - COMANDA O PROXIMO BIT...
         SELECIONADO : Bool := TRUE;   // 1=MOTOR SELECIONADO
         JOG : Bool;   // 1=JOG
         MARCHA : Bool;   // 1=MARCHA
         FRENTE_REVERSAO : Bool;   // SENTIDO DE ROTAÇÃO DO MOTOR // 0=FRENTE - 1=REVERSÃO
         RESERVA_5 : Byte;   // RESERVA
         RESERVA_6 : Byte;   // RESERVA
         RESERVA_30 : Bool;   // RESERVA
         RESERVA_31 : Bool;   // RESERVA
         RESERVA_32 : Bool;   // RESERVA
         RESERVA_33 : Bool;   // RESERVA
         RESERVA_34 : Bool;   // RESERVA
         RESERVA_35 : Bool;   // RESERVA
         STATUS_DRIVER : Bool := TRUE;   // BIT AUXILIAR DE STATUS DO INVERSOR DE FREQUENCIA - 1=OK
         DESBLOQUEIO_DRIVER : Bool;   // BIT AUXILIAR DE DESBLOQUEIO DO INVERSOR DE FREQÊNCIA
      END_STRUCT;
      REFERENCIAS : Struct   // REFERÊNCIAS
         BASE : Real;   // BASE SEM ACC/DEC
         FINAL : Real;   // FINAL COM ACC/DEC
         TAXA : Real := -1.0;   // TAXA - -20...20%
         RESERVA_20 : Real;   // RESERVA
         RESERVA_24 : Real;   // RESERVA
         RESERVA_28 : Real;   // RESERVA
         RESERVA_32 : Real;   // RESERVA
         RESERVA_36 : Real;   // RESERVA
         RESERVA_40 : Real;   // RESERVA
         RESERVA_44 : Real;   // RESERVA
         VELOCIDADE_MAXIMA : Real := 8000.0;   // VELOCIDADE MAXIMA - 0=0M/MIN // 10.000=100M/MIN - CALCULADO AUTOMÁTICAMENTE
      END_STRUCT;
   END_VAR
BEGIN
END_DATA_BLOCK

DATA_BLOCK "DB SECADEIRA2"   // DB22
TITLE = Automation Pack Automação Indl. e Com. Ltda.
{ S7_Optimized_Access := 'FALSE' }
AUTHOR : THALLES
FAMILY : TRAÇÃO
NAME : LINHA1
VERSION : 0.1
// Cliente: Texima S/A Ind. de Máquinas
// Cliente Final: Cia. Fiação e Tecidos Santo Antonio.
// Máquina: Linha 1 DENIN - O.S.: 24.626
   VAR
      ALARMES : Struct   // ALARMES
         PROTECAO_INVERSOR : Bool;   // ALARME DE NIVEL ALTO - PROTEÇÃO DO INVERSOR DE FREQUENCIA
         RESERVA_01 : Bool;   // ALARME DE NIVEL ALTO - RESERVA
         BALANCA_INFERIOR : Bool;   // ALARME DE NIVEL ALTO - BALANÇA INFERIOR
         BALANCA_SUPERIOR : Bool;   // ALARME DE NIVEL ALTO - BALANÇA SUPERIOR
         RESERVA_10 : Byte;   // ALARME DE NIVEL ALTO - RESERVA
         RESERVA_20 : Byte;   // ALARME DE NIVEL BAIXO - RESERVA
         RESERVA_30 : Byte;   // ALARME DE NIVEL BAIXO - RESERVA
      END_STRUCT;
      COMANDOS : Struct   // COMANDOS
         SELECAO : Bool;   // COMANDO PARA SELEÇÃO "ON/OFF" - COMANDA O PROXIMO BIT...
         SELECIONADO : Bool := TRUE;   // 1=MOTOR SELECIONADO
         JOG : Bool;   // 1=JOG
         MARCHA : Bool;   // 1=MARCHA
         FRENTE_REVERSAO : Bool;   // SENTIDO DE ROTAÇÃO DO MOTOR // 0=FRENTE - 1=REVERSÃO
         RESERVA_5 : Byte;   // RESERVA
         RESERVA_6 : Byte;   // RESERVA
         RESERVA_30 : Bool;   // RESERVA
         RESERVA_31 : Bool;   // RESERVA
         RESERVA_32 : Bool;   // RESERVA
         RESERVA_33 : Bool;   // RESERVA
         RESERVA_34 : Bool;   // RESERVA
         RESERVA_35 : Bool;   // RESERVA
         STATUS_DRIVER : Bool := TRUE;   // BIT AUXILIAR DE STATUS DO INVERSOR DE FREQUENCIA - 1=OK
         DESBLOQUEIO_DRIVER : Bool;   // BIT AUXILIAR DE DESBLOQUEIO DO INVERSOR DE FREQÊNCIA
      END_STRUCT;
      REFERENCIAS : Struct   // REFERÊNCIAS
         BASE : Real;   // BASE SEM ACC/DEC
         FINAL : Real;   // FINAL COM ACC/DEC
         CORRECAO : Real;   // CORRECAO BALANCA
         BALANCA : Real := 100.0;   // POSIÇÃO DA BALANÇA - -100...0...100%
         GANHO_BALANCA : Real;   // GANHO DA BALAÇA - 10%...30% - REFERENTE A VELOCIDADE MÁXIMA DA MÁQUINA
         RESERVA_28 : Real;   // RESERVA
         RESERVA_32 : Real;   // RESERVA
         RESERVA_36 : Real;   // RESERVA
         RESERVA_40 : Real;   // RESERVA
         RESERVA_44 : Real;   // RESERVA
         VELOCIDADE_MAXIMA : Real := 8000.0;   // VELOCIDADE MAXIMA - 0=0M/MIN // 10.000=100M/MIN - CALCULADO AUTOMÁTICAMENTE
      END_STRUCT;
   END_VAR
BEGIN
END_DATA_BLOCK

DATA_BLOCK "DB SECADEIRA3"   // DB23
TITLE = Automation Pack Automação Indl. e Com. Ltda.
{ S7_Optimized_Access := 'FALSE' }
AUTHOR : THALLES
FAMILY : TRAÇÃO
NAME : LINHA1
VERSION : 0.1
// Cliente: Texima S/A Ind. de Máquinas
// Cliente Final: Cia. Fiação e Tecidos Santo Antonio.
// Máquina: Linha 1 DENIN - O.S.: 24.626
   VAR
      ALARMES : Struct   // ALARMES
         PROTECAO_INVERSOR : Bool;   // ALARME DE NIVEL ALTO - PROTEÇÃO DO INVERSOR DE FREQUENCIA
         RESERVA_01 : Bool;   // ALARME DE NIVEL ALTO - RESERVA
         BALANCA_INFERIOR : Bool;   // ALARME DE NIVEL ALTO - BALANÇA INFERIOR
         BALANCA_SUPERIOR : Bool := TRUE;   // ALARME DE NIVEL ALTO - BALANÇA SUPERIOR
         RESERVA_10 : Byte;   // ALARME DE NIVEL ALTO - RESERVA
         RESERVA_20 : Byte;   // ALARME DE NIVEL BAIXO - RESERVA
         RESERVA_30 : Byte;   // ALARME DE NIVEL BAIXO - RESERVA
      END_STRUCT;
      COMANDOS : Struct   // COMANDOS
         SELECAO : Bool;   // COMANDO PARA SELEÇÃO "ON/OFF" - COMANDA O PROXIMO BIT...
         SELECIONADO : Bool := TRUE;   // 1=MOTOR SELECIONADO
         JOG : Bool;   // 1=JOG
         MARCHA : Bool;   // 1=MARCHA
         FRENTE_REVERSAO : Bool;   // SENTIDO DE ROTAÇÃO DO MOTOR // 0=FRENTE - 1=REVERSÃO
         RESERVA_5 : Byte;   // RESERVA
         RESERVA_6 : Byte;   // RESERVA
         RESERVA_30 : Bool;   // RESERVA
         RESERVA_31 : Bool;   // RESERVA
         RESERVA_32 : Bool;   // RESERVA
         RESERVA_33 : Bool;   // RESERVA
         RESERVA_34 : Bool;   // RESERVA
         RESERVA_35 : Bool;   // RESERVA
         STATUS_DRIVER : Bool := TRUE;   // BIT AUXILIAR DE STATUS DO INVERSOR DE FREQUENCIA - 1=OK
         DESBLOQUEIO_DRIVER : Bool;   // BIT AUXILIAR DE DESBLOQUEIO DO INVERSOR DE FREQÊNCIA
      END_STRUCT;
      REFERENCIAS : Struct   // REFERÊNCIAS
         BASE : Real;   // BASE SEM ACC/DEC
         FINAL : Real;   // FINAL COM ACC/DEC
         CORRECAO : Real;   // CORRECAO BALANCA
         BALANCA : Real := -95.07075;   // POSIÇÃO DA BALANÇA - -100...0...100%
         GANHO_BALANCA : Real;   // GANHO DA BALAÇA - 10%...30% - REFERENTE A VELOCIDADE MÁXIMA DA MÁQUINA
         RESERVA_28 : Real;   // RESERVA
         RESERVA_32 : Real;   // RESERVA
         RESERVA_36 : Real;   // RESERVA
         RESERVA_40 : Real;   // RESERVA
         RESERVA_44 : Real;   // RESERVA
         VELOCIDADE_MAXIMA : Real := 8000.0;   // VELOCIDADE MAXIMA - 0=0M/MIN // 10.000=100M/MIN - CALCULADO AUTOMÁTICAMENTE
      END_STRUCT;
   END_VAR
BEGIN
END_DATA_BLOCK

DATA_BLOCK "DB SECADEIRA4"   // DB24
TITLE = Automation Pack Automação Indl. e Com. Ltda.
{ S7_Optimized_Access := 'FALSE' }
AUTHOR : THALLES
FAMILY : TRAÇÃO
NAME : LINHA1
VERSION : 0.1
// Cliente: Texima S/A Ind. de Máquinas
// Cliente Final: Cia. Fiação e Tecidos Santo Antonio.
// Máquina: Linha 1 DENIN - O.S.: 24.626
   VAR
      ALARMES : Struct   // ALARMES
         PROTECAO_INVERSOR : Bool;   // ALARME DE NIVEL ALTO - PROTEÇÃO DO INVERSOR DE FREQUENCIA
         RESERVA_01 : Bool;   // ALARME DE NIVEL ALTO - RESERVA
         BALANCA_INFERIOR : Bool;   // ALARME DE NIVEL ALTO - BALANÇA INFERIOR
         BALANCA_SUPERIOR : Bool := TRUE;   // ALARME DE NIVEL ALTO - BALANÇA SUPERIOR
         RESERVA_10 : Byte;   // ALARME DE NIVEL ALTO - RESERVA
         RESERVA_20 : Byte;   // ALARME DE NIVEL BAIXO - RESERVA
         RESERVA_30 : Byte;   // ALARME DE NIVEL BAIXO - RESERVA
      END_STRUCT;
      COMANDOS : Struct   // COMANDOS
         SELECAO : Bool;   // COMANDO PARA SELEÇÃO "ON/OFF" - COMANDA O PROXIMO BIT...
         SELECIONADO : Bool := TRUE;   // 1=MOTOR SELECIONADO
         JOG : Bool;   // 1=JOG
         MARCHA : Bool;   // 1=MARCHA
         FRENTE_REVERSAO : Bool;   // SENTIDO DE ROTAÇÃO DO MOTOR // 0=FRENTE - 1=REVERSÃO
         RESERVA_5 : Byte;   // RESERVA
         RESERVA_6 : Byte;   // RESERVA
         RESERVA_30 : Bool;   // RESERVA
         RESERVA_31 : Bool;   // RESERVA
         RESERVA_32 : Bool;   // RESERVA
         RESERVA_33 : Bool;   // RESERVA
         RESERVA_34 : Bool;   // RESERVA
         RESERVA_35 : Bool;   // RESERVA
         STATUS_DRIVER : Bool := TRUE;   // BIT AUXILIAR DE STATUS DO INVERSOR DE FREQUENCIA - 1=OK
         DESBLOQUEIO_DRIVER : Bool;   // BIT AUXILIAR DE DESBLOQUEIO DO INVERSOR DE FREQÊNCIA
      END_STRUCT;
      REFERENCIAS : Struct   // REFERÊNCIAS
         BASE : Real;   // BASE SEM ACC/DEC
         FINAL : Real;   // FINAL COM ACC/DEC
         CORRECAO : Real;   // CORRECAO BALANCA
         BALANCA : Real := 100.0;   // POSIÇÃO DA BALANÇA - -100...0...100%
         GANHO_BALANCA : Real;   // GANHO DA BALAÇA - 10%...30% - REFERENTE A VELOCIDADE MÁXIMA DA MÁQUINA
         RESERVA_28 : Real;   // RESERVA
         RESERVA_32 : Real;   // RESERVA
         RESERVA_36 : Real;   // RESERVA
         RESERVA_40 : Real;   // RESERVA
         RESERVA_44 : Real;   // RESERVA
         VELOCIDADE_MAXIMA : Real := 8000.0;   // VELOCIDADE MAXIMA - 0=0M/MIN // 10.000=100M/MIN - CALCULADO AUTOMÁTICAMENTE
      END_STRUCT;
   END_VAR
BEGIN
END_DATA_BLOCK

DATA_BLOCK "DB PUXADOR_JOTA_SAIDA"   // DB25
TITLE = Automation Pack Automação Indl. e Com. Ltda.
{ S7_Optimized_Access := 'FALSE' }
AUTHOR : THALLES
FAMILY : TRAÇÃO
NAME : LINHA1
VERSION : 0.1
// Cliente: Texima S/A Ind. de Máquinas
// Cliente Final: Cia. Fiação e Tecidos Santo Antonio.
// Máquina: Linha 1 DENIN - O.S.: 24.626
   VAR
      ALARMES : Struct   // ALARMES
         PROTECAO_INVERSOR : Bool;   // ALARME DE NIVEL ALTO - PROTEÇÃO DO INVERSOR DE FREQUENCIA
         RESERVA_01 : Bool;   // ALARME DE NIVEL ALTO - RESERVA
         BALANCA_INFERIOR : Bool;   // ALARME DE NIVEL ALTO - BALANÇA INFERIOR
         BALANCA_SUPERIOR : Bool := TRUE;   // ALARME DE NIVEL ALTO - BALANÇA SUPERIOR
         RESERVA_10 : Byte;   // ALARME DE NIVEL ALTO - RESERVA
         RESERVA_20 : Byte;   // ALARME DE NIVEL BAIXO - RESERVA
         RESERVA_30 : Byte;   // ALARME DE NIVEL BAIXO - RESERVA
      END_STRUCT;
      COMANDOS : Struct   // COMANDOS
         SELECAO : Bool;   // COMANDO PARA SELEÇÃO "ON/OFF" - COMANDA O PROXIMO BIT...
         SELECIONADO : Bool := TRUE;   // 1=MOTOR SELECIONADO
         JOG : Bool;   // 1=JOG
         MARCHA : Bool;   // 1=MARCHA
         FRENTE_REVERSAO : Bool;   // SENTIDO DE ROTAÇÃO DO MOTOR // 0=FRENTE - 1=REVERSÃO
         RESERVA_5 : Byte;   // RESERVA
         RESERVA_6 : Byte;   // RESERVA
         RESERVA_30 : Bool;   // RESERVA
         RESERVA_31 : Bool;   // RESERVA
         RESERVA_32 : Bool;   // RESERVA
         RESERVA_33 : Bool;   // RESERVA
         RESERVA_34 : Bool;   // RESERVA
         RESERVA_35 : Bool;   // RESERVA
         STATUS_DRIVER : Bool := TRUE;   // BIT AUXILIAR DE STATUS DO INVERSOR DE FREQUENCIA - 1=OK
         DESBLOQUEIO_DRIVER : Bool;   // BIT AUXILIAR DE DESBLOQUEIO DO INVERSOR DE FREQÊNCIA
      END_STRUCT;
      REFERENCIAS : Struct   // REFERÊNCIAS
         BASE : Real;   // BASE SEM ACC/DEC
         FINAL : Real;   // FINAL COM ACC/DEC
         CORRECAO : Real;   // CORRECAO BALANCA
         BALANCA : Real := 100.0;   // POSIÇÃO DA BALANÇA - -100...0...100%
         GANHO_BALANCA : Real;   // GANHO DA BALAÇA - 10%...30% - REFERENTE A VELOCIDADE MÁXIMA DA MÁQUINA
         RESERVA_28 : Real;   // RESERVA
         RESERVA_32 : Real;   // RESERVA
         RESERVA_36 : Real;   // RESERVA
         RESERVA_40 : Real;   // RESERVA
         RESERVA_44 : Real;   // RESERVA
         VELOCIDADE_MAXIMA : Real := 8000.0;   // VELOCIDADE MAXIMA - 0=0M/MIN // 10.000=100M/MIN - CALCULADO AUTOMÁTICAMENTE
      END_STRUCT;
   END_VAR
BEGIN
END_DATA_BLOCK

DATA_BLOCK "DB ENROLADOR_GIGANTE"   // DB26
TITLE = Automation Pack Automação Indl. e Com. Ltda.
{ S7_Optimized_Access := 'FALSE' }
AUTHOR : THALLES
FAMILY : TRAÇÃO
NAME : LINHA1
VERSION : 0.1
// Cliente: Texima S/A Ind. de Máquinas
// Cliente Final: Cia. Fiação e Tecidos Santo Antonio.
// Máquina: Linha 1 DENIN - O.S.: 24.626
   VAR
      ALARMES : Struct   // ALARMES
         PROTECAO_INVERSOR : Bool;   // ALARME DE NIVEL ALTO - PROTEÇÃO DO INVERSOR DE FREQUENCIA
         RESERVA_01 : Bool;   // ALARME DE NIVEL ALTO - RESERVA
         BALANCA_INFERIOR : Bool;   // ALARME DE NIVEL ALTO - BALANÇA INFERIOR
         BALANCA_SUPERIOR : Bool;   // ALARME DE NIVEL ALTO - BALANÇA SUPERIOR
         RESERVA_10 : Byte;   // ALARME DE NIVEL ALTO - RESERVA
         RESERVA_20 : Byte;   // ALARME DE NIVEL BAIXO - RESERVA
         RESERVA_30 : Byte;   // ALARME DE NIVEL BAIXO - RESERVA
      END_STRUCT;
      COMANDOS : Struct   // COMANDOS
         SELECAO : Bool;   // COMANDO PARA SELEÇÃO "ON/OFF" - COMANDA O PROXIMO BIT...
         SELECIONADO : Bool;   // 1=MOTOR SELECIONADO
         JOG : Bool;   // 1= JOG
         MARCHA : Bool := TRUE;   // 1=MARCHA
         FRENTE_REVERSAO : Bool;   // SENTIDO DE ROTAÇÃO DO MOTOR // 0=FRENTE - 1=REVERSÃO
         RESERVA_45 : Bool;   // RESERVA
         RESERVA_46 : Bool := TRUE;   // RESERVA
         RESERVA_47 : Bool;   // RESERVA
         SINC_INDEP : Bool := TRUE;   // TIPO DE CONTROLE // 0=SINCRONIZADO - 1=INDEPENDENTE
         TROCA_ROLO : Bool;   // 1=MODO TROCA ROLO ATIVO
         CONTROLE_INDEPENDENTE : Bool := TRUE;   // 1=CONTROLE INDEPENDENTE ATIVO
         SINCRONISMO : Bool;   // AUXILIAR - REALIZA O SINCRONISMO COM A MÁQUINA APOS O TROCA ROLO
         JOG_SUPER : Bool;   // RESERVA
         RESERVA_55 : Bool;   // RESERVA
         RESERVA_56 : Bool;   // RESERVA
         RESERVA_57 : Bool;   // RESERVA
         RESERVA_60 : Byte;   // RESERVA
         RESERVA_70 : Bool;   // RESERVA
         RESERVA_71 : Bool;   // RESERVA
         RESERVA_72 : Bool;   // RESERVA
         RESERVA_73 : Bool;   // RESERVA
         RESERVA_74 : Bool;   // RESERVA
         RESERVA_75 : Bool;   // RESERVA
         STATUS_DRIVER : Bool := TRUE;   // BIT AUXILIAR DE STATUS DO INVERSOR DE FREQUENCIA - 1=OK
         DESBLOQUEIO_DRIVER : Bool;   // BIT AUXILIAR DE DESBLOQUEIO DO INVERSOR DE FREQÊNCIA
      END_STRUCT;
      REFERENCIAS : Struct   // REFERÊNCIAS
         BASE : Real;   // BASE SEM ACC/DEC
         FINAL : Real := 16#5224_FBE5_0200_D037;   // FINAL COM ACC/DEC
         CORRECAO : Real;   // CORRECAO BALANCA
         BALANCA : Real := 100.0;   // POSIÇÃO DA BALANÇA - -100...0...100%
         GANHO_BALANCA : Real;   // GANHO DA BALAÇA - 10%...30% - REFERENTE A VELOCIDADE MÁXIMA DA MÁQUINA
         INDEPENDENTE : Real;   // REFERÊNCIA INDEPENDENTE - AJUSTADA PELO POTENCIÔMETRO NA REMOTA DO PUXADOR
         RESERVA_320 : Real;   // RESERVA
         RESERVA_360 : Real;   // RESERVA
         RESERVA_400 : Real;   // RESERVA
         RESERVA_440 : Real;   // RESERVA
         VELOCIDADE_MAXIMA : Real := 8000.0;   // VELOCIDADE MAXIMA - 0=0M/MIN // 10.000=100M/MIN - CALCULADO AUTOMÁTICAMENTE
      END_STRUCT;
   END_VAR
BEGIN
END_DATA_BLOCK

DATA_BLOCK "DB BALANCA 1"   // DB30
{ S7_Optimized_Access := 'FALSE' }
AUTHOR : THALLES
FAMILY : BALANCA
VERSION : 0.1
// stored: InstanceOfName FB BALANCA
"FB BALANCA"
BEGIN
END_DATA_BLOCK

DATA_BLOCK "DB BALANCA 2"   // DB31
{ S7_Optimized_Access := 'FALSE' }
AUTHOR : THALLES
FAMILY : BALANCA
VERSION : 0.1
// stored: InstanceOfName FB BALANCA
"FB BALANCA"
BEGIN
END_DATA_BLOCK

DATA_BLOCK "DB BALANCA 3"   // DB32
{ S7_Optimized_Access := 'FALSE' }
AUTHOR : THALLES
FAMILY : BALANCA
VERSION : 0.1
// stored: InstanceOfName FB BALANCA
"FB BALANCA"
BEGIN
END_DATA_BLOCK

DATA_BLOCK "DB BALANCA 4"   // DB33
{ S7_Optimized_Access := 'FALSE' }
AUTHOR : THALLES
FAMILY : BALANCA
VERSION : 0.1
// stored: InstanceOfName FB BALANCA
"FB BALANCA"
BEGIN
END_DATA_BLOCK

DATA_BLOCK "DB BALANCA 5"   // DB34
{ S7_Optimized_Access := 'FALSE' }
AUTHOR : THALLES
FAMILY : BALANCA
VERSION : 0.1
// stored: InstanceOfName FB BALANCA
"FB BALANCA"
BEGIN
END_DATA_BLOCK

DATA_BLOCK "DB BALANCA 6"   // DB35
{ S7_Optimized_Access := 'FALSE' }
AUTHOR : THALLES
FAMILY : BALANCA
VERSION : 0.1
// stored: InstanceOfName FB BALANCA
"FB BALANCA"
BEGIN
END_DATA_BLOCK

DATA_BLOCK "DB BALANCA 7"   // DB36
{ S7_Optimized_Access := 'FALSE' }
AUTHOR : THALLES
FAMILY : BALANCA
VERSION : 0.1
// stored: InstanceOfName FB BALANCA
"FB BALANCA"
BEGIN
END_DATA_BLOCK

DATA_BLOCK "DB BALANCA 8"   // DB37
{ S7_Optimized_Access := 'FALSE' }
AUTHOR : THALLES
FAMILY : BALANCA
VERSION : 0.1
// stored: InstanceOfName FB BALANCA
"FB BALANCA"
BEGIN
END_DATA_BLOCK

DATA_BLOCK "DB BALANCA 9"   // DB38
{ S7_Optimized_Access := 'FALSE' }
AUTHOR : THALLES
FAMILY : BALANCA
VERSION : 0.1
// stored: InstanceOfName FB BALANCA
"FB BALANCA"
BEGIN
END_DATA_BLOCK

DATA_BLOCK "DB BALANCA 10"   // DB39
{ S7_Optimized_Access := 'FALSE' }
AUTHOR : THALLES
FAMILY : BALANCA
VERSION : 0.1
// stored: InstanceOfName FB BALANCA
"FB BALANCA"
BEGIN
END_DATA_BLOCK

DATA_BLOCK "DB BALANCA 11"   // DB40
{ S7_Optimized_Access := 'FALSE' }
AUTHOR : THALLES
FAMILY : BALANCA
VERSION : 0.1
// stored: InstanceOfName FB BALANCA
"FB BALANCA"
BEGIN
END_DATA_BLOCK

DATA_BLOCK "DB BALANCA 12"   // DB41
{ S7_Optimized_Access := 'FALSE' }
AUTHOR : THALLES
FAMILY : BALANCA
VERSION : 0.1
// stored: InstanceOfName FB BALANCA
"FB BALANCA"
BEGIN
END_DATA_BLOCK

DATA_BLOCK "DB BALANCA 13"   // DB42
{ S7_Optimized_Access := 'FALSE' }
AUTHOR : THALLES
FAMILY : BALANCA
VERSION : 0.1
// stored: InstanceOfName FB BALANCA
"FB BALANCA"
BEGIN
END_DATA_BLOCK

DATA_BLOCK "DB CELULA EXTRACTA 1"   // DB43
{ S7_Optimized_Access := 'FALSE' }
AUTHOR : THALLES
VERSION : 0.1
// stored: InstanceOfName CELULA_CARGA
"CELULA_CARGA"
BEGIN
END_DATA_BLOCK

DATA_BLOCK "DB CELULA EXTRACTA 2"   // DB44
{ S7_Optimized_Access := 'FALSE' }
AUTHOR : THALLES
VERSION : 0.1
// stored: InstanceOfName CELULA_CARGA
"CELULA_CARGA"
BEGIN
END_DATA_BLOCK

DATA_BLOCK "DB VALORES TRANSMITIDOS"   // DB200
TITLE = Automation Pack Automação Indl. e Com. Ltda.
{ S7_Optimized_Access := 'FALSE' }
AUTHOR : ANDERSON
FAMILY : OS:24626
NAME : SANFOR
VERSION : 0.1
// Cliente: Texima S/A Ind. de Máquinas
// Cliente Final: Cia. Fiação e Tecidos Santo Antonio.
// Máquina: Sanforizadeira da Linha Integrada 1 - O.S.: 24.626
   VAR
      VARIAVEIS_COMPARTILHADAS : Struct   // VARIÁVEIS COMUNS AS DUAS MÁQUINAS
         DIGITAIS : Struct   // SINAIS DIGITAIS
            LIGA_MAQUINA : Bool;   // BIT DO BOTÃO DE LIGA MÁQUINA
            DESLIGA_MAQUINA : Bool := TRUE;   // BIT DO BOTÃO DE DESLIGA MÁQUINA
            EMERGENCIA_GERAL : Bool := TRUE;   // BIT DO BOTÃO DE EMERGÊNCIA GERAL
            JOG_GERAL : Bool;   // BIT DO BOTÃO DE JOG GERAL
            TRAVA_BALANCA : Bool;   // BIT DO BOTÃO DE TRAVA BALANÇA
            DESTRAVA_ALARME : Bool;   // BIT DO BOTÃO DE DESTRAVA ALARME
            PRESSOSTATO_MAQUINA : Bool := TRUE;   // BIT DO PRESSOSTATO DA MÁQUINA
            ALARME_ALTO : Bool := TRUE;   // BIT QUE INDICA QUE ALGUM ALARME DE NIVEL ALTO FOI GERADO
            ALARME_BAIXO : Bool := TRUE;   // BIT QUE INDICA QUE ALGUM ALARME DE NIVEL BAIXO FOI GERADO
            BALANCA_FORA_POSICAO : Bool;   // BIT QUE INDICA ALARME DAS BALANÇAS - 1=INDICAÇÃO DE BALANÇA FORA DE POSIÇÃO
            MARCHA : Bool;   // BIT QUE INDICA ESTADO DA MÁQUINA - 1=MÁQUINA LIGADA
            AUX_MARCHA : Bool;   // BIT QUE INDICA ESTADO DO AUXILIAR DO COMANDO DE LIGA MAQUINA
            MOTOR_SELECIONADO : Bool := TRUE;   // BIT QUE INDICA SELEÇÃO DOS MOTORES - 1=ALGUM MOTOR DE TRAÇÃO ESTÁ SELECIONADO
         END_STRUCT;
      END_STRUCT;
      VARIAVEIS_LINHA : Struct   // VARIÁVEIS RECEBIDAS PELA SANFOR DA A LINHA
         DIGITAIS : Struct   // SINAIS DIGITAIS
            RESERVA2_0 : Bool;   // RESERVA
         END_STRUCT;
         ANALOGICAS : Struct   // SINAIS ANALÓGICOS
            REFERENCIA_BASE_LINHA : Real := 800.0;   // REFERÊNCIA BASE DA LINHA SEM ACC/DEC
            POSICAO_REAL_BALANCA : Int := 28236;   // POSIÇÃO REAL DA BALANÇA DE SINCRONISMO - VALOR ANALÓGICO
         END_STRUCT;
      END_STRUCT;
   END_VAR
BEGIN
END_DATA_BLOCK

DATA_BLOCK "DB VALORES RECEBIDOS"   // DB201
TITLE = Automation Pack Automação Indl. e Com. Ltda.
{ S7_Optimized_Access := 'FALSE' }
AUTHOR : ANDERSON
FAMILY : OS:24626
NAME : SANFOR
VERSION : 0.1
// Cliente: Texima S/A Ind. de Máquinas
// Cliente Final: Cia. Fiação e Tecidos Santo Antonio.
// Máquina: Sanforizadeira da Linha Integrada 1 - O.S.: 24.626
   VAR
      VARIAVEIS_COMPARTILHADAS : Struct   // VARIÁVEIS COMUNS AS DUAS MÁQUINAS
         DIGITAIS : Struct   // SINAIS DIGITAIS
            LIGA_MAQUINA : Bool;   // BIT DO BOTÃO DE LIGA MÁQUINA
            DESLIGA_MAQUINA : Bool := TRUE;   // BIT DO BOTÃO DE DESLIGA MÁQUINA
            EMERGENCIA_GERAL : Bool := TRUE;   // BIT DO BOTÃO DE EMERGÊNCIA GERAL
            JOG_GERAL : Bool;   // BIT DO BOTÃO DE JOG GERAL
            TRAVA_BALANCA : Bool;   // BIT DO BOTÃO DE TRAVA BALANÇA
            DESTRAVA_ALARME : Bool;   // BIT DO BOTÃO DE DESTRAVA ALARME
            PRESSOSTATO_MAQUINA : Bool := TRUE;   // BIT DO PRESSOSTATO DA MÁQUINA
            ALARME_ALTO : Bool;   // BIT QUE INDICA QUE ALGUM ALARME DE NIVEL ALTO FOI GERADO
            ALARME_BAIXO : Bool;   // BIT QUE INDICA QUE ALGUM ALARME DE NIVEL BAIXO FOI GERADO
            BALANCA_FORA_POSICAO : Bool;   // BIT QUE INDICA ALARME DAS BALANÇAS - 1=INDICAÇÃO DE BALANÇA FORA DE POSIÇÃO
            MARCHA : Bool;   // BIT QUE INDICA ESTADO DA MÁQUINA - 1=MÁQUINA LIGADA
            AUX_MARCHA : Bool;   // BIT QUE INDICA ESTADO DO AUXILIAR DO COMANDO DE LIGA MAQUINA
            MOTOR_SELECIONADO : Bool := TRUE;   // BIT QUE INDICA SELEÇÃO DOS MOTORES - 1=ALGUM MOTOR DE TRAÇÃO ESTÁ SELECIONADO
            BIT_ACIONAMNETO_ALRM : Bool;   // BIT QUE ACIONA A CAMPANHIA DE ALARME DA MAQUINA
         END_STRUCT;
      END_STRUCT;
      VARIAVEIS_SANFOR : Struct   // VARIÁVEIS ENVIADAS PELA SANFOR PARA A LINHA
         DIGITAIS : Struct   // SINAIS DIGITAIS
            MAIS_VELOCIDADE : Bool;   // BIT DO BOTÃO DE MAIS VELOCIDADE
            MENOS_VELOCIDADE : Bool;   // BIT DO BOTÃO DE MENOS VELOCIDADE
            MODO_INDEP_SINC : Bool;   // BIT DO MODO DE OPERAÇÃO DAS MÁQUINAS // 0=INDEPENDENTE - 1=SINCRONIZADO
         END_STRUCT;
         ANALOGICAS : Struct   // SINAIS ANALÓGICOS
            PER_VMS_TORRE_SECAGEM : Int;   // VALOR MANIPULADO DE SAÍDA - TORRE DE SECAGEM - PERIFÉRICO
         END_STRUCT;
      END_STRUCT;
   END_VAR
BEGIN
END_DATA_BLOCK

FUNCTION_BLOCK "FB BALANCA"   // FB30, LAD
{ S7_Optimized_Access := 'FALSE' }
AUTHOR : THALLES
FAMILY : BALANCA
NAME : LINHA1
VERSION : 0.1
   VAR_INPUT
      INPUT_MAX : Real;
      INPUT_MIN : Real;
      REFERENCIA_BASE : Real;
      CORRECAO_MAXIMA : Real;
      BALANCA : Int;
      MODO : Bool;
   END_VAR
   VAR_OUTPUT
      CORRECAO : Real;
   END_VAR
   VAR
      MR0 : Real;
      MR1 : Real;
      MR2 : Real;
      MR3 : Real;
      MR4 : Real;
      MR5 : Real;
      MDI0 : DInt;
   END_VAR
BEGIN

REGION Network 1
   // CONVERTE INTEIRO EM REAL
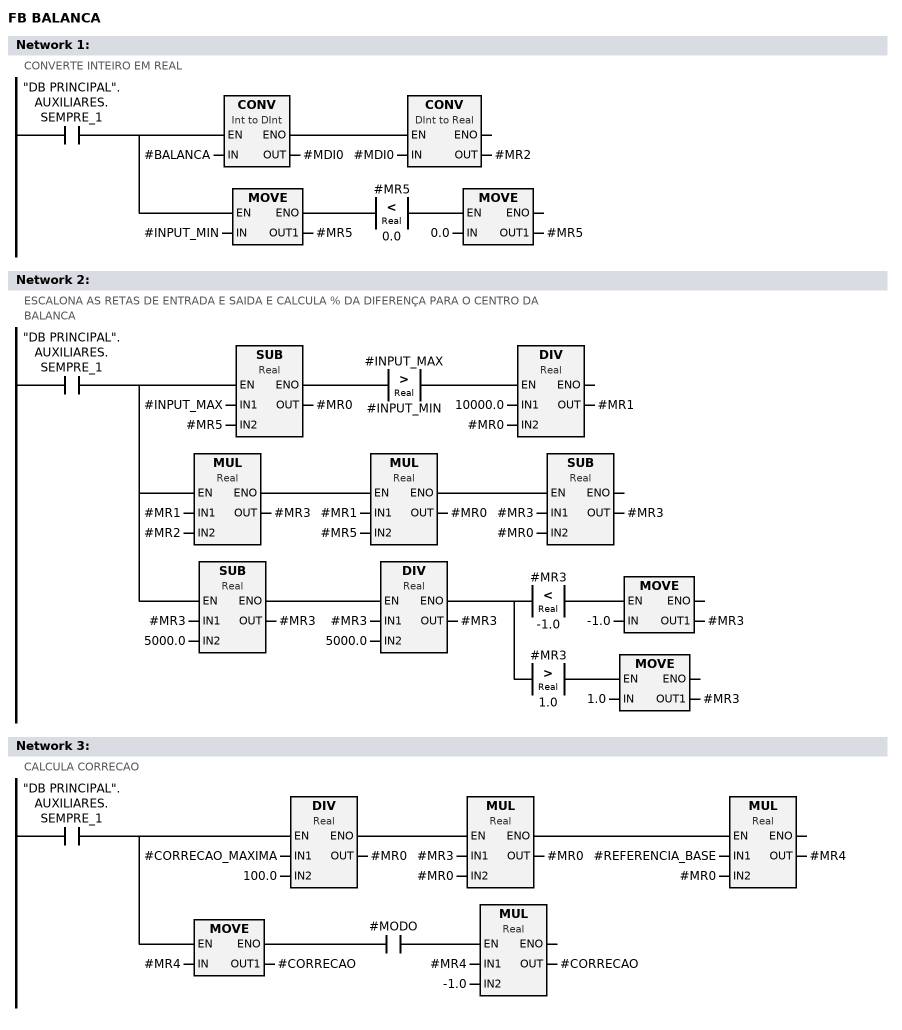
   RUNG wire#powerrail
      Contact( "DB PRINCIPAL".AUXILIARES.SEMPRE_1 )
      wire#w1
      { S7_Templates := "[SrcType := Int, DestType := DInt]"; S7_GenerateENO := "TRUE" } Convert(in := #BALANCA, out => #MDI0)
      { S7_Templates := "[SrcType := DInt, DestType := Real]"; S7_GenerateENO := "TRUE" } Convert(in := #MDI0, out => #MR2)
   END_RUNG
   RUNG wire#w1
      { S7_GenerateENO := "TRUE" } Move(in := #INPUT_MIN, out1 => #MR5)
      { S7_Templates := "SrcType := Real" } LT_Contact(in1 := #MR5, in2 := 0.0)
      { S7_GenerateENO := "TRUE" } Move(in := 0.0, out1 => #MR5)
   END_RUNG
   // the same network as SCL:
   // ENO of a box is taken as its EN; it also drops when the box reports an error
   IF "DB PRINCIPAL".AUXILIARES.SEMPRE_1 THEN
       #MDI0 := INT_TO_DINT(#BALANCA);
       #MR2 := DINT_TO_REAL(#MDI0);
       #MR5 := #INPUT_MIN;
   END_IF;
   IF "DB PRINCIPAL".AUXILIARES.SEMPRE_1 AND (#MR5 < 0.0) THEN #MR5 := 0.0; END_IF;
END_REGION

REGION Network 2
   // ESCALONA AS RETAS DE ENTRADA E SAIDA E CALCULA % DA DIFERENÇA PARA O CENTRO DA 
   // BALANCA
   RUNG wire#powerrail
      Contact( "DB PRINCIPAL".AUXILIARES.SEMPRE_1 )
      wire#w1
      { S7_Templates := "SrcType := Real"; S7_GenerateENO := "TRUE" } Sub(in1 := #INPUT_MAX, in2 := #MR5, out => #MR0)
      { S7_Templates := "SrcType := Real" } GT_Contact(in1 := #INPUT_MAX, in2 := #INPUT_MIN)
      { S7_Templates := "SrcType := Real"; S7_GenerateENO := "TRUE" } Div(in1 := 10000.0, in2 := #MR0, out => #MR1)
   END_RUNG
   RUNG wire#w1
      { S7_Templates := "SrcType := Real"; S7_GenerateENO := "TRUE" } Mul(in1 := #MR1, in2 := #MR2, out => #MR3)
      { S7_Templates := "SrcType := Real"; S7_GenerateENO := "TRUE" } Mul(in1 := #MR1, in2 := #MR5, out => #MR0)
      { S7_Templates := "SrcType := Real"; S7_GenerateENO := "TRUE" } Sub(in1 := #MR3, in2 := #MR0, out => #MR3)
   END_RUNG
   RUNG wire#w1
      { S7_Templates := "SrcType := Real"; S7_GenerateENO := "TRUE" } Sub(in1 := #MR3, in2 := 5000.0, out => #MR3)
      { S7_Templates := "SrcType := Real"; S7_GenerateENO := "TRUE" } Div(in1 := #MR3, in2 := 5000.0, out => #MR3)
      wire#w2
      { S7_Templates := "SrcType := Real" } LT_Contact(in1 := #MR3, in2 := -1.0)
      { S7_GenerateENO := "TRUE" } Move(in := -1.0, out1 => #MR3)
   END_RUNG
   RUNG wire#w2
      { S7_Templates := "SrcType := Real" } GT_Contact(in1 := #MR3, in2 := 1.0)
      { S7_GenerateENO := "TRUE" } Move(in := 1.0, out1 => #MR3)
   END_RUNG
   // the same network as SCL:
   // ENO of a box is taken as its EN; it also drops when the box reports an error
   IF "DB PRINCIPAL".AUXILIARES.SEMPRE_1 THEN #MR0 := #INPUT_MAX - #MR5; END_IF;
   IF "DB PRINCIPAL".AUXILIARES.SEMPRE_1 AND (#INPUT_MAX > #INPUT_MIN) THEN #MR1 := 10000.0 / #MR0; END_IF;
   IF "DB PRINCIPAL".AUXILIARES.SEMPRE_1 THEN
       #MR3 := #MR1 * #MR2;
       #MR0 := #MR1 * #MR5;
       #MR3 := #MR3 - #MR0;
       #MR3 := #MR3 - 5000.0;
       #MR3 := #MR3 / 5000.0;
   END_IF;
   IF "DB PRINCIPAL".AUXILIARES.SEMPRE_1 AND (#MR3 < (-1.0)) THEN #MR3 := -1.0; END_IF;
   IF "DB PRINCIPAL".AUXILIARES.SEMPRE_1 AND (#MR3 > 1.0) THEN #MR3 := 1.0; END_IF;
END_REGION

REGION Network 3
   // CALCULA CORRECAO
   RUNG wire#powerrail
      Contact( "DB PRINCIPAL".AUXILIARES.SEMPRE_1 )
      wire#w1
      { S7_Templates := "SrcType := Real"; S7_GenerateENO := "TRUE" } Div(in1 := #CORRECAO_MAXIMA, in2 := 100.0, out => #MR0)
      { S7_Templates := "SrcType := Real"; S7_GenerateENO := "TRUE" } Mul(in1 := #MR3, in2 := #MR0, out => #MR0)
      { S7_Templates := "SrcType := Real"; S7_GenerateENO := "TRUE" } Mul(in1 := #REFERENCIA_BASE, in2 := #MR0, out => #MR4)
   END_RUNG
   RUNG wire#w1
      { S7_GenerateENO := "TRUE" } Move(in := #MR4, out1 => #CORRECAO)
      Contact( #MODO )
      { S7_Templates := "SrcType := Real"; S7_GenerateENO := "TRUE" } Mul(in1 := #MR4, in2 := -1.0, out => #CORRECAO)
   END_RUNG
   // the same network as SCL:
   // ENO of a box is taken as its EN; it also drops when the box reports an error
   IF "DB PRINCIPAL".AUXILIARES.SEMPRE_1 THEN
       #MR0 := #CORRECAO_MAXIMA / 100.0;
       #MR0 := #MR3 * #MR0;
       #MR4 := #REFERENCIA_BASE * #MR0;
       #CORRECAO := #MR4;
   END_IF;
   IF "DB PRINCIPAL".AUXILIARES.SEMPRE_1 AND #MODO THEN #CORRECAO := #MR4 * (-1.0); END_IF;
END_REGION
END_FUNCTION_BLOCK

FUNCTION_BLOCK "CELULA_CARGA"   // FB50, LAD
{ S7_Optimized_Access := 'FALSE' }
AUTHOR : THALLES
VERSION : 0.1
   VAR_INPUT
      TRIGGER : Bool;
      CELULA : Int;
      SETPOINT : Real;
      COR_MAX : Real;
      VELOCIDADE_BASE : Real;
   END_VAR
   VAR_OUTPUT
      CORRECAO : Real;
      CELULA_REAL : Real;
   END_VAR
   VAR
      MI0 : Real;
      MI1 : Real;
      MI2 : Real;
      MI3 : Real;
      MI4 : Real;
      MEDIA : Real;
      AUX_DI : DInt;
      AUX_R : Real;
      FATOR : Real;
      AUX_R2 : Real;
      W1 : Int;
      borda : Bool;
      calcula : Bool;
   END_VAR
   VAR_TEMP   // added for the SCL form of the ladder/FBD networks
      _w1 : Bool;
   END_VAR
BEGIN

REGION Network 1
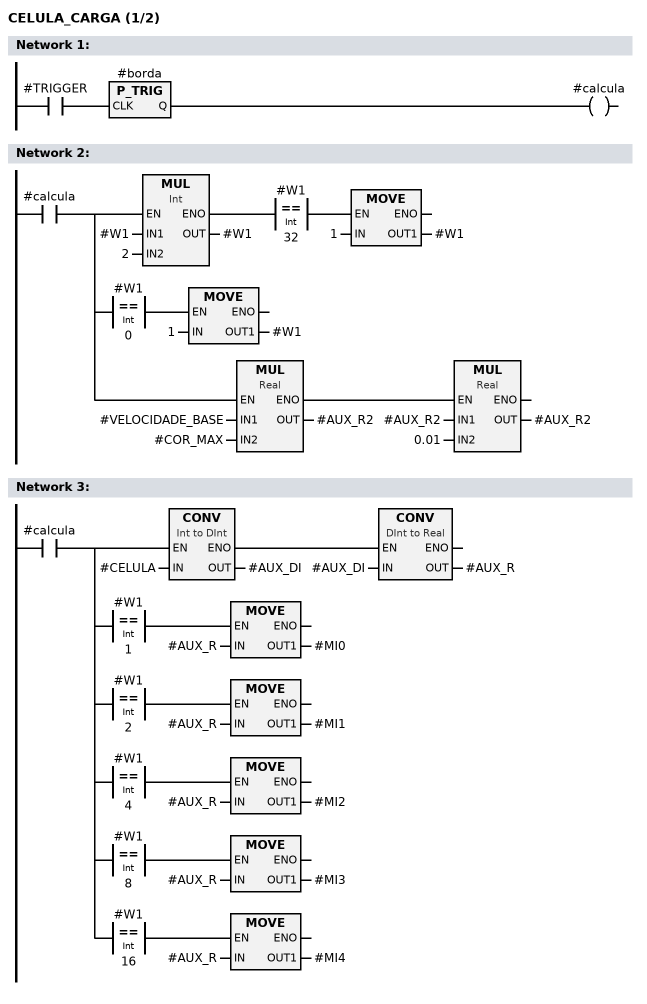
   RUNG wire#powerrail
      Contact( #TRIGGER )
      P_Trig( #borda )
      Coil( #calcula )
   END_RUNG
   // the same network as SCL:
   #_w1 := #TRIGGER AND NOT #borda;   // rising edge
   #borda := #TRIGGER;
   #calcula := #_w1;
END_REGION

REGION Network 2
   RUNG wire#powerrail
      Contact( #calcula )
      wire#w1
      { S7_Templates := "SrcType := Int"; S7_GenerateENO := "TRUE" } Mul(in1 := #W1, in2 := 2, out => #W1)
      { S7_Templates := "SrcType := Int" } EQ_Contact(in1 := #W1, in2 := 32)
      { S7_GenerateENO := "TRUE" } Move(in := 1, out1 => #W1)
   END_RUNG
   RUNG wire#w1
      { S7_Templates := "SrcType := Int" } EQ_Contact(in1 := #W1, in2 := 0)
      { S7_GenerateENO := "TRUE" } Move(in := 1, out1 => #W1)
   END_RUNG
   RUNG wire#w1
      { S7_Templates := "SrcType := Real"; S7_GenerateENO := "TRUE" } Mul(in1 := #VELOCIDADE_BASE, in2 := #COR_MAX, out => #AUX_R2)
      { S7_Templates := "SrcType := Real"; S7_GenerateENO := "TRUE" } Mul(in1 := #AUX_R2, in2 := 0.01, out => #AUX_R2)
   END_RUNG
   // the same network as SCL:
   // ENO of a box is taken as its EN; it also drops when the box reports an error
   IF #calcula THEN #W1 := #W1 * 2; END_IF;
   IF #calcula AND (#W1 = 32) THEN #W1 := 1; END_IF;
   IF #calcula AND (#W1 = 0) THEN #W1 := 1; END_IF;
   IF #calcula THEN
       #AUX_R2 := #VELOCIDADE_BASE * #COR_MAX;
       #AUX_R2 := #AUX_R2 * 0.01;
   END_IF;
END_REGION

REGION Network 3
   RUNG wire#powerrail
      Contact( #calcula )
      wire#w1
      { S7_Templates := "[SrcType := Int, DestType := DInt]"; S7_GenerateENO := "TRUE" } Convert(in := #CELULA, out => #AUX_DI)
      { S7_Templates := "[SrcType := DInt, DestType := Real]"; S7_GenerateENO := "TRUE" } Convert(in := #AUX_DI, out => #AUX_R)
   END_RUNG
   RUNG wire#w1
      { S7_Templates := "SrcType := Int" } EQ_Contact(in1 := #W1, in2 := 1)
      { S7_GenerateENO := "TRUE" } Move(in := #AUX_R, out1 => #MI0)
   END_RUNG
   RUNG wire#w1
      { S7_Templates := "SrcType := Int" } EQ_Contact(in1 := #W1, in2 := 2)
      { S7_GenerateENO := "TRUE" } Move(in := #AUX_R, out1 => #MI1)
   END_RUNG
   RUNG wire#w1
      { S7_Templates := "SrcType := Int" } EQ_Contact(in1 := #W1, in2 := 4)
      { S7_GenerateENO := "TRUE" } Move(in := #AUX_R, out1 => #MI2)
   END_RUNG
   RUNG wire#w1
      { S7_Templates := "SrcType := Int" } EQ_Contact(in1 := #W1, in2 := 8)
      { S7_GenerateENO := "TRUE" } Move(in := #AUX_R, out1 => #MI3)
   END_RUNG
   RUNG wire#w1
      { S7_Templates := "SrcType := Int" } EQ_Contact(in1 := #W1, in2 := 16)
      { S7_GenerateENO := "TRUE" } Move(in := #AUX_R, out1 => #MI4)
   END_RUNG
   // the same network as SCL:
   // ENO of a box is taken as its EN; it also drops when the box reports an error
   IF #calcula THEN
       #AUX_DI := INT_TO_DINT(#CELULA);
       #AUX_R := DINT_TO_REAL(#AUX_DI);
   END_IF;
   IF #calcula AND (#W1 = 1) THEN #MI0 := #AUX_R; END_IF;
   IF #calcula AND (#W1 = 2) THEN #MI1 := #AUX_R; END_IF;
   IF #calcula AND (#W1 = 4) THEN #MI2 := #AUX_R; END_IF;
   IF #calcula AND (#W1 = 8) THEN #MI3 := #AUX_R; END_IF;
   IF #calcula AND (#W1 = 16) THEN #MI4 := #AUX_R; END_IF;
END_REGION

REGION Network 4
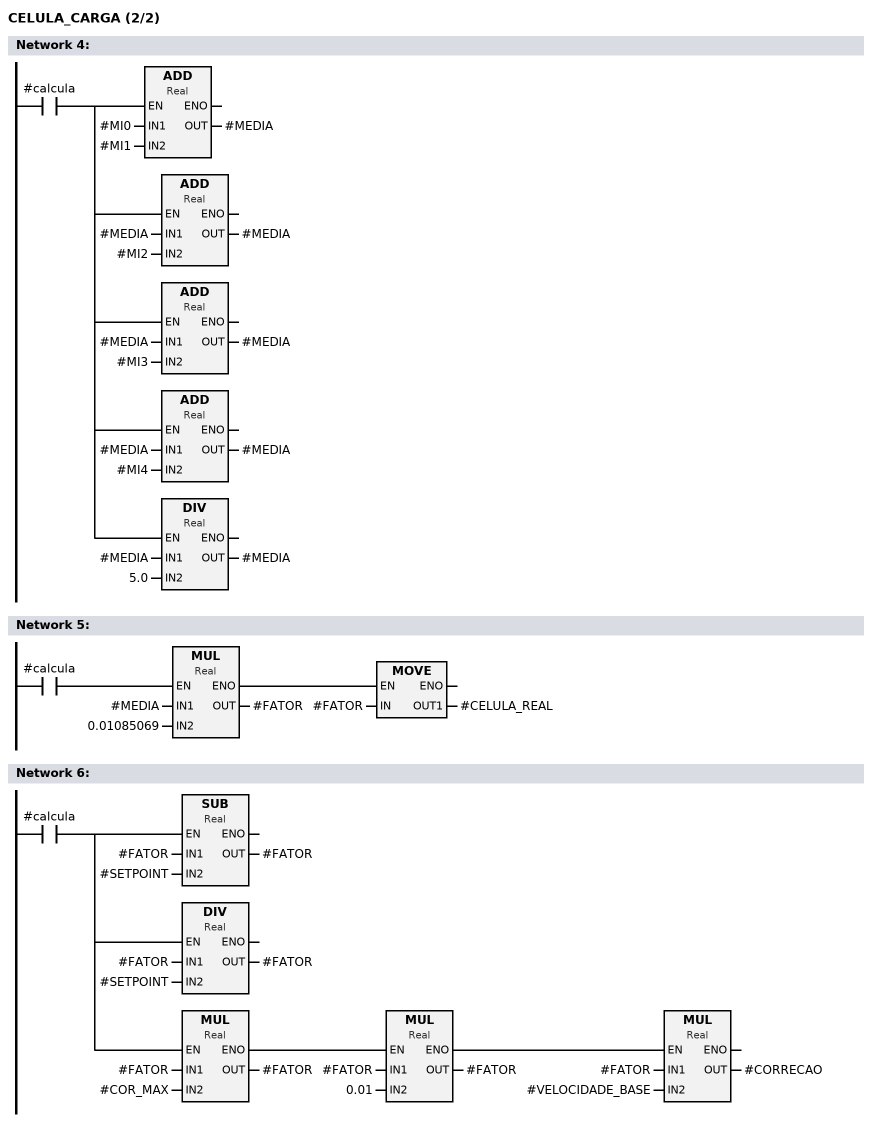
   RUNG wire#powerrail
      Contact( #calcula )
      wire#w1
      { S7_Templates := "SrcType := Real"; S7_GenerateENO := "TRUE" } Add(in1 := #MI0, in2 := #MI1, out => #MEDIA)
   END_RUNG
   RUNG wire#w1
      { S7_Templates := "SrcType := Real"; S7_GenerateENO := "TRUE" } Add(in1 := #MEDIA, in2 := #MI2, out => #MEDIA)
   END_RUNG
   RUNG wire#w1
      { S7_Templates := "SrcType := Real"; S7_GenerateENO := "TRUE" } Add(in1 := #MEDIA, in2 := #MI3, out => #MEDIA)
   END_RUNG
   RUNG wire#w1
      { S7_Templates := "SrcType := Real"; S7_GenerateENO := "TRUE" } Add(in1 := #MEDIA, in2 := #MI4, out => #MEDIA)
   END_RUNG
   RUNG wire#w1
      { S7_Templates := "SrcType := Real"; S7_GenerateENO := "TRUE" } Div(in1 := #MEDIA, in2 := 5.0, out => #MEDIA)
   END_RUNG
   // the same network as SCL:
   IF #calcula THEN
       #MEDIA := #MI0 + #MI1;
       #MEDIA := #MEDIA + #MI2;
       #MEDIA := #MEDIA + #MI3;
       #MEDIA := #MEDIA + #MI4;
       #MEDIA := #MEDIA / 5.0;
   END_IF;
END_REGION

REGION Network 5
   RUNG wire#powerrail
      Contact( #calcula )
      { S7_Templates := "SrcType := Real"; S7_GenerateENO := "TRUE" } Mul(in1 := #MEDIA, in2 := 0.01085069, out => #FATOR)
      { S7_GenerateENO := "TRUE" } Move(in := #FATOR, out1 => #CELULA_REAL)
   END_RUNG
   // the same network as SCL:
   // ENO of a box is taken as its EN; it also drops when the box reports an error
   IF #calcula THEN
       #FATOR := #MEDIA * 0.01085069;
       #CELULA_REAL := #FATOR;
   END_IF;
END_REGION

